KUKA KRL program: f1_Kuka_APT206T02S06.SRC

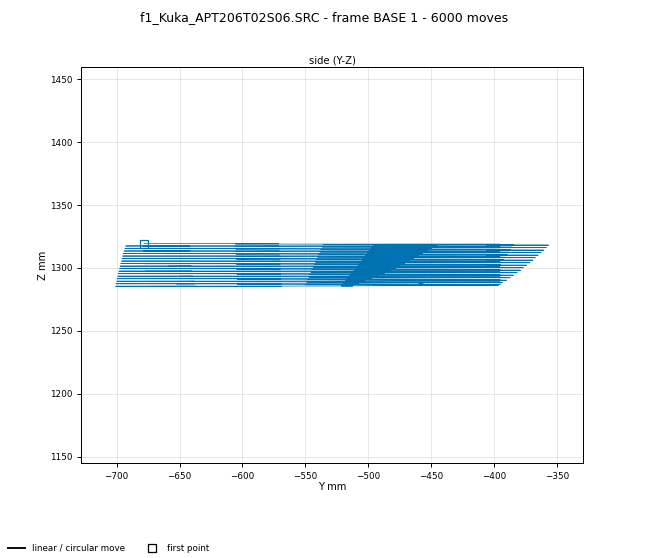
[picture p0: tool path of f1_Kuka_APT206T02S06.SRC in frame BASE 1, 6000 of 6001 moves have a stored position in this frame; points joined in program order, loops and branches not executed]
&ACCESS RVP
&REL 2
&PARAM TEMPLATE = C:\KRC\Roboter\Template\vorgabe
&PARAM EDITMASK = *
DEF f1_Kuka_APT206T02S06()


;FOLD INI;%{PE}%V3.2.0,%MKUKATPBASIS,%CINIT,%VCOMMON,%P
  ;FOLD BAS INI;%{E}%V3.2.0,%MKUKATPBASIS,%CINIT,%VINIT,%P
    GLOBAL INTERRUPT DECL 3 WHEN $STOPMESS==TRUE DO IR_STOPM ( )
    INTERRUPT ON 3
    BAS (#INITMOV,0 )
  ;ENDFOLD (BAS INI)
  ;FOLD USER INI;%{E}%V3.2.0,%MKUKATPUSER,%CINIT,%VINIT,%P
    ;Make your modifications here
  ;ENDFOLD (USER INI)
;ENDFOLD (INI)


;*** Make Null PTP Move
  PTP $pos_act

;*** Auto Load The Correct TOOL Data
  $tool=tool_data[2]

;*** Auto Load The Correct BASE Data
  $base=base_data[1]

  $ADVANCE = 5

;*** Restate Last Velocity
MMPM(30000.0)
SetRPM(8000)
LIN {X -0.383,Y -678.241,Z 1319.360,A 0.000,B 0.000,C 90.000,E1 100.782} C_DIS
LIN {X 0.191,Y -677.668,Z 1319.357,A 0.000,B 0.000,C 90.000,E1 100.254} C_DIS
LIN {X -0.027,Y -676.905,Z 1319.354,A 0.000,B 0.000,C 90.000,E1 99.792} C_DIS
LIN {X -0.134,Y -675.753,Z 1319.352,A 0.000,B 0.000,C 90.000,E1 99.321} C_DIS
LIN {X 0.307,Y -674.318,Z 1319.349,A 0.000,B 0.000,C 90.000,E1 98.803} C_DIS
LIN {X 0.076,Y -672.539,Z 1319.346,A 0.000,B 0.000,C 90.000,E1 98.341} C_DIS
LIN {X -0.071,Y -670.513,Z 1319.344,A 0.000,B 0.000,C 90.000,E1 97.871} C_DIS
LIN {X 0.337,Y -668.279,Z 1319.341,A 0.000,B 0.000,C 90.000,E1 97.352} C_DIS
LIN {X 0.069,Y -665.838,Z 1319.338,A 0.000,B 0.000,C 90.000,E1 96.891} C_DIS
LIN {X -0.309,Y -662.485,Z 1319.335,A 0.000,B 0.000,C 90.000,E1 96.315} C_DIS
LIN {X 0.043,Y -659.568,Z 1319.332,A 0.000,B 0.000,C 90.000,E1 95.796} C_DIS
LIN {X -0.281,Y -656.447,Z 1319.330,A 0.000,B 0.000,C 90.000,E1 95.334} C_DIS
LIN {X 0.072,Y -653.986,Z 1319.328,A 0.000,B 0.000,C 90.000,E1 94.935} C_DIS
LIN {X 0.254,Y -649.358,Z 1319.324,A 0.000,B 0.000,C 90.000,E1 94.302} C_DIS
LIN {X -0.138,Y -645.441,Z 1319.321,A 0.000,B 0.000,C 90.000,E1 93.841} C_DIS
LIN {X -0.068,Y -640.049,Z 1319.318,A 0.000,B 0.000,C 90.000,E1 93.212} C_DIS
LIN {X 0.118,Y -635.523,Z 1319.315,A 0.000,B 0.000,C 90.000,E1 92.694} C_DIS
LIN {X 0.245,Y -630.728,Z 1319.312,A 0.000,B 0.000,C 90.000,E1 92.178} C_DIS
LIN {X -0.245,Y -624.406,Z 1319.309,A 0.000,B 0.000,C 90.000,E1 91.604} C_DIS
LIN {X 0.064,Y -617.770,Z 1319.306,A 0.000,B 0.000,C 90.000,E1 90.974} C_DIS
LIN {X 0.019,Y -614.904,Z 1319.304,A 0.000,B 0.000,C 90.000,E1 90.745} C_DIS
LIN {X -0.082,Y -609.367,Z 1319.302,A 0.000,B 0.000,C 90.000,E1 90.344} C_DIS
LIN {X -0.088,Y -602.730,Z 1319.300,A 0.000,B 0.000,C 90.000,E1 89.943} C_DIS
LIN {X -0.187,Y -595.944,Z 1319.298,A 0.000,B 0.000,C 90.000,E1 89.599} C_DIS
LIN {X 0.165,Y -588.900,Z 1319.296,A 0.000,B 0.000,C 90.000,E1 89.255} C_DIS
LIN {X -0.024,Y -576.693,Z 1319.293,A 0.000,B 0.000,C 90.000,E1 88.797} C_DIS
LIN {X 0.193,Y -573.915,Z 1319.292,A 0.000,B 0.000,C 90.000,E1 88.625} C_DIS
LIN {X -0.066,Y -572.871,Z 1319.292,A 0.000,B 0.000,C 90.000,E1 88.568} C_DIS
LIN {X -0.103,Y -571.871,Z 1319.291,A 0.000,B 0.000,C 90.000,E1 88.453} C_DIS
LIN {X -0.146,Y -571.844,Z 1319.291,A 0.000,B 0.000,C 90.000,E1 88.453} C_DIS
LIN {X 0.218,Y -571.236,Z 1319.289,A 0.000,B 0.000,C 90.000,E1 88.051} C_DIS
LIN {X 0.134,Y -571.299,Z 1319.287,A 0.000,B 0.000,C 90.000,E1 87.650} C_DIS
LIN {X -0.010,Y -573.083,Z 1319.276,A 0.000,B 0.000,C 90.000,E1 85.755} C_DIS
LIN {X 0.263,Y -575.744,Z 1319.263,A 0.000,B 0.000,C 90.000,E1 83.280} C_DIS
LIN {X 0.201,Y -577.711,Z 1319.254,A 0.000,B 0.000,C 90.000,E1 81.659} C_DIS
LIN {X -0.044,Y -579.300,Z 1319.246,A 0.000,B 0.000,C 90.000,E1 80.330} C_DIS
LIN {X -0.175,Y -580.807,Z 1319.239,A 0.000,B 0.000,C 90.000,E1 78.993} C_DIS
LIN {X 0.169,Y -581.938,Z 1319.233,A 0.000,B 0.000,C 90.000,E1 77.881} C_DIS
LIN {X 0.193,Y -583.136,Z 1319.225,A 0.000,B 0.000,C 90.000,E1 76.533} C_DIS
LIN {X 0.043,Y -584.329,Z 1319.216,A 0.000,B 0.000,C 90.000,E1 74.936} C_DIS
LIN {X 0.076,Y -585.456,Z 1319.207,A 0.000,B 0.000,C 90.000,E1 73.323} C_DIS
LIN {X 0.230,Y -586.154,Z 1319.202,A 0.000,B 0.000,C 90.000,E1 72.236} C_DIS
LIN {X -0.261,Y -587.227,Z 1319.193,A 0.000,B 0.000,C 90.000,E1 70.678} C_DIS
LIN {X 0.165,Y -588.716,Z 1319.179,A 0.000,B 0.000,C 90.000,E1 68.230} C_DIS
LIN {X -0.209,Y -589.764,Z 1319.170,A 0.000,B 0.000,C 90.000,E1 66.666} C_DIS
LIN {X -0.020,Y -590.895,Z 1319.161,A 0.000,B 0.000,C 90.000,E1 65.049} C_DIS
LIN {X -0.038,Y -592.401,Z 1319.150,A 0.000,B 0.000,C 90.000,E1 62.922} C_DIS
LIN {X -0.001,Y -593.510,Z 1319.142,A 0.000,B 0.000,C 90.000,E1 61.591} C_DIS
LIN {X 0.096,Y -594.716,Z 1319.135,A 0.000,B 0.000,C 90.000,E1 60.255} C_DIS
LIN {X -0.078,Y -596.020,Z 1319.127,A 0.000,B 0.000,C 90.000,E1 58.948} C_DIS
LIN {X -0.312,Y -597.969,Z 1319.117,A 0.000,B 0.000,C 90.000,E1 57.120} C_DIS
LIN {X -0.311,Y -599.376,Z 1319.110,A 0.000,B 0.000,C 90.000,E1 55.801} C_DIS
LIN {X -0.284,Y -600.719,Z 1319.103,A 0.000,B 0.000,C 90.000,E1 54.482} C_DIS
LIN {X 0.114,Y -601.929,Z 1319.095,A 0.000,B 0.000,C 90.000,E1 53.130} C_DIS
LIN {X 0.055,Y -603.065,Z 1319.088,A 0.000,B 0.000,C 90.000,E1 51.823} C_DIS
LIN {X -0.244,Y -603.807,Z 1319.082,A 0.000,B 0.000,C 90.000,E1 50.803} C_DIS
LIN {X 0.106,Y -604.726,Z 1319.075,A 0.000,B 0.000,C 90.000,E1 49.461} C_DIS
LIN {X -0.043,Y -605.108,Z 1319.071,A 0.000,B 0.000,C 90.000,E1 48.690} C_DIS
LIN {X 0.066,Y -605.351,Z 1319.065,A 0.000,B 0.000,C 90.000,E1 47.634} C_DIS
LIN {X -0.002,Y -605.572,Z 1319.055,A 0.000,B 0.000,C 90.000,E1 45.810} C_DIS
LIN {X 0.276,Y -605.578,Z 1319.050,A 0.000,B 0.000,C 90.000,E1 45.000} C_DIS
LIN {X -0.029,Y -605.233,Z 1319.042,A 0.000,B 0.000,C 90.000,E1 43.461} C_DIS
LIN {X -0.319,Y -604.735,Z 1319.033,A 0.000,B 0.000,C 90.000,E1 41.919} C_DIS
LIN {X -0.415,Y -604.251,Z 1319.026,A 0.000,B 0.000,C 90.000,E1 40.620} C_DIS
LIN {X -0.018,Y -603.365,Z 1319.015,A 0.000,B 0.000,C 90.000,E1 38.749} C_DIS
LIN {X -0.317,Y -602.720,Z 1319.010,A 0.000,B 0.000,C 90.000,E1 37.729} C_DIS
LIN {X -0.036,Y -602.043,Z 1319.005,A 0.000,B 0.000,C 90.000,E1 36.916} C_DIS
LIN {X -0.126,Y -601.079,Z 1319.001,A 0.000,B 0.000,C 90.000,E1 36.137} C_DIS
LIN {X -0.086,Y -599.082,Z 1318.993,A 0.000,B 0.000,C 90.000,E1 34.818} C_DIS
LIN {X -0.077,Y -596.688,Z 1318.986,A 0.000,B 0.000,C 90.000,E1 33.499} C_DIS
LIN {X 0.269,Y -594.911,Z 1318.982,A 0.000,B 0.000,C 90.000,E1 32.673} C_DIS
LIN {X -0.331,Y -592.256,Z 1318.976,A 0.000,B 0.000,C 90.000,E1 31.671} C_DIS
LIN {X -0.233,Y -590.717,Z 1318.973,A 0.000,B 0.000,C 90.000,E1 31.131} C_DIS
LIN {X -0.261,Y -588.078,Z 1318.968,A 0.000,B 0.000,C 90.000,E1 30.335} C_DIS
LIN {X -0.314,Y -585.030,Z 1318.964,A 0.000,B 0.000,C 90.000,E1 29.539} C_DIS
LIN {X 0.236,Y -582.780,Z 1318.961,A 0.000,B 0.000,C 90.000,E1 28.949} C_DIS
LIN {X 0.121,Y -579.160,Z 1318.957,A 0.000,B 0.000,C 90.000,E1 28.153} C_DIS
LIN {X 0.202,Y -574.998,Z 1318.952,A 0.000,B 0.000,C 90.000,E1 27.334} C_DIS
LIN {X 0.073,Y -571.204,Z 1318.948,A 0.000,B 0.000,C 90.000,E1 26.668} C_DIS
LIN {X 0.163,Y -567.135,Z 1318.944,A 0.000,B 0.000,C 90.000,E1 25.976} C_DIS
LIN {X 0.219,Y -562.748,Z 1318.941,A 0.000,B 0.000,C 90.000,E1 25.283} C_DIS
LIN {X -0.269,Y -557.850,Z 1318.937,A 0.000,B 0.000,C 90.000,E1 24.643} C_DIS
LIN {X 0.063,Y -553.956,Z 1318.934,A 0.000,B 0.000,C 90.000,E1 24.079} C_DIS
LIN {X 0.002,Y -548.431,Z 1318.930,A 0.000,B 0.000,C 90.000,E1 23.387} C_DIS
LIN {X 0.018,Y -543.698,Z 1318.927,A 0.000,B 0.000,C 90.000,E1 22.823} C_DIS
LIN {X 0.077,Y -536.444,Z 1318.922,A 0.000,B 0.000,C 90.000,E1 21.972} C_DIS
LIN {X 0.048,Y -531.264,Z 1318.919,A 0.000,B 0.000,C 90.000,E1 21.408} C_DIS
LIN {X 0.199,Y -522.283,Z 1318.914,A 0.000,B 0.000,C 90.000,E1 20.429} C_DIS
LIN {X 0.149,Y -511.815,Z 1318.908,A 0.000,B 0.000,C 90.000,E1 19.341} C_DIS
LIN {X 0.057,Y -502.681,Z 1318.902,A 0.000,B 0.000,C 90.000,E1 18.417} C_DIS
LIN {X -0.001,Y -491.518,Z 1318.896,A 0.000,B 0.000,C 90.000,E1 17.330} C_DIS
LIN {X -0.041,Y -483.324,Z 1318.892,A 0.000,B 0.000,C 90.000,E1 16.551} C_DIS
LIN {X 0.178,Y -474.592,Z 1318.887,A 0.000,B 0.000,C 90.000,E1 15.717} C_DIS
LIN {X 0.167,Y -464.311,Z 1318.882,A 0.000,B 0.000,C 90.000,E1 14.773} C_DIS
LIN {X 0.215,Y -446.791,Z 1318.873,A 0.000,B 0.000,C 90.000,E1 13.119} C_DIS
LIN {X 0.151,Y -424.007,Z 1318.860,A 0.000,B 0.000,C 90.000,E1 10.782} C_DIS
LIN {X 0.086,Y -406.860,Z 1318.850,A 0.000,B 0.000,C 90.000,E1 8.916} C_DIS
LIN {X -0.204,Y -398.311,Z 1318.844,A 0.000,B 0.000,C 90.000,E1 7.992} C_DIS
LIN {X -0.085,Y -395.321,Z 1318.842,A 0.000,B 0.000,C 90.000,E1 7.530} C_DIS
LIN {X -0.124,Y -395.315,Z 1318.842,A 0.000,B 0.000,C 90.000,E1 7.530} C_DIS
LIN {X 0.155,Y -395.949,Z 1318.841,A 0.000,B 0.000,C 90.000,E1 7.352} C_DIS
LIN {X 0.118,Y -395.998,Z 1318.841,A 0.000,B 0.000,C 90.000,E1 7.352} C_DIS
LIN {X -0.054,Y -399.469,Z 1318.839,A 0.000,B 0.000,C 90.000,E1 7.068} C_DIS
LIN {X 0.042,Y -405.000,Z 1318.837,A 0.000,B 0.000,C 90.000,E1 6.663} C_DIS
LIN {X 0.063,Y -409.735,Z 1318.835,A 0.000,B 0.000,C 90.000,E1 6.372} C_DIS
LIN {X 0.004,Y -417.825,Z 1318.833,A 0.000,B 0.000,C 90.000,E1 5.853} C_DIS
LIN {X 0.038,Y -424.124,Z 1318.830,A 0.000,B 0.000,C 90.000,E1 5.391} C_DIS
LIN {X -0.173,Y -430.359,Z 1318.827,A 0.000,B 0.000,C 90.000,E1 4.935} C_DIS
LIN {X -0.043,Y -439.367,Z 1318.823,A 0.000,B 0.000,C 90.000,E1 4.131} C_DIS
LIN {X -0.035,Y -443.739,Z 1318.821,A 0.000,B 0.000,C 90.000,E1 3.726} C_DIS
LIN {X 0.021,Y -449.647,Z 1318.818,A 0.000,B 0.000,C 90.000,E1 3.154} C_DIS
LIN {X 0.047,Y -455.368,Z 1318.814,A 0.000,B 0.000,C 90.000,E1 2.579} C_DIS
LIN {X -0.123,Y -460.898,Z 1318.811,A 0.000,B 0.000,C 90.000,E1 2.007} C_DIS
LIN {X 0.217,Y -467.528,Z 1318.807,A 0.000,B 0.000,C 90.000,E1 1.203} C_DIS
LIN {X -0.216,Y -472.449,Z 1318.803,A 0.000,B 0.000,C 90.000,E1 0.630} C_DIS
LIN {X 0.000,Y -476.981,Z 1318.800,A 0.000,B 0.000,C 90.000,E1 360.000} C_DIS
LIN {X 0.121,Y -481.653,Z 1318.796,A 0.000,B 0.000,C 90.000,E1 359.312} C_DIS
LIN {X -0.103,Y -486.586,Z 1318.792,A 0.000,B 0.000,C 90.000,E1 358.568} C_DIS
LIN {X 0.222,Y -491.172,Z 1318.788,A 0.000,B 0.000,C 90.000,E1 357.764} C_DIS
LIN {X 0.081,Y -495.438,Z 1318.784,A 0.000,B 0.000,C 90.000,E1 357.020} C_DIS
LIN {X -0.179,Y -498.630,Z 1318.780,A 0.000,B 0.000,C 90.000,E1 356.445} C_DIS
LIN {X -0.041,Y -503.078,Z 1318.775,A 0.000,B 0.000,C 90.000,E1 355.527} C_DIS
LIN {X -0.048,Y -506.551,Z 1318.771,A 0.000,B 0.000,C 90.000,E1 354.780} C_DIS
LIN {X -0.078,Y -511.007,Z 1318.765,A 0.000,B 0.000,C 90.000,E1 353.742} C_DIS
LIN {X -0.226,Y -513.361,Z 1318.762,A 0.000,B 0.000,C 90.000,E1 353.166} C_DIS
LIN {X 0.122,Y -516.546,Z 1318.757,A 0.000,B 0.000,C 90.000,E1 352.243} C_DIS
LIN {X -0.006,Y -519.467,Z 1318.752,A 0.000,B 0.000,C 90.000,E1 351.376} C_DIS
LIN {X -0.022,Y -521.276,Z 1318.749,A 0.000,B 0.000,C 90.000,E1 350.792} C_DIS
LIN {X -0.103,Y -523.788,Z 1318.744,A 0.000,B 0.000,C 90.000,E1 349.926} C_DIS
LIN {X -0.068,Y -526.011,Z 1318.739,A 0.000,B 0.000,C 90.000,E1 349.050} C_DIS
LIN {X 0.018,Y -528.682,Z 1318.733,A 0.000,B 0.000,C 90.000,E1 347.881} C_DIS
LIN {X 0.225,Y -530.374,Z 1318.728,A 0.000,B 0.000,C 90.000,E1 346.992} C_DIS
LIN {X -0.184,Y -531.781,Z 1318.723,A 0.000,B 0.000,C 90.000,E1 346.172} C_DIS
LIN {X 0.104,Y -533.446,Z 1318.717,A 0.000,B 0.000,C 90.000,E1 344.991} C_DIS
LIN {X -0.145,Y -534.384,Z 1318.712,A 0.000,B 0.000,C 90.000,E1 344.157} C_DIS
LIN {X 0.130,Y -535.065,Z 1318.707,A 0.000,B 0.000,C 90.000,E1 343.268} C_DIS
LIN {X 0.055,Y -535.458,Z 1318.702,A 0.000,B 0.000,C 90.000,E1 342.417} C_DIS
LIN {X -0.177,Y -535.659,Z 1318.698,A 0.000,B 0.000,C 90.000,E1 341.583} C_DIS
LIN {X -0.239,Y -535.454,Z 1318.693,A 0.000,B 0.000,C 90.000,E1 340.732} C_DIS
LIN {X -0.094,Y -534.784,Z 1318.687,A 0.000,B 0.000,C 90.000,E1 339.571} C_DIS
LIN {X 0.128,Y -534.219,Z 1318.683,A 0.000,B 0.000,C 90.000,E1 338.975} C_DIS
LIN {X 0.240,Y -533.293,Z 1318.679,A 0.000,B 0.000,C 90.000,E1 338.103} C_DIS
LIN {X -0.053,Y -532.872,Z 1318.677,A 0.000,B 0.000,C 90.000,E1 337.847} C_DIS
LIN {X 0.051,Y -531.324,Z 1318.672,A 0.000,B 0.000,C 90.000,E1 336.975} C_DIS
LIN {X -0.157,Y -528.693,Z 1318.666,A 0.000,B 0.000,C 90.000,E1 335.845} C_DIS
LIN {X 0.205,Y -527.147,Z 1318.663,A 0.000,B 0.000,C 90.000,E1 335.229} C_DIS
LIN {X -0.235,Y -524.541,Z 1318.658,A 0.000,B 0.000,C 90.000,E1 334.409} C_DIS
LIN {X 0.059,Y -519.924,Z 1318.650,A 0.000,B 0.000,C 90.000,E1 332.922} C_DIS
LIN {X 0.023,Y -515.240,Z 1318.641,A 0.000,B 0.000,C 90.000,E1 331.463} C_DIS
LIN {X 0.037,Y -511.177,Z 1318.635,A 0.000,B 0.000,C 90.000,E1 330.284} C_DIS
LIN {X -0.085,Y -508.003,Z 1318.630,A 0.000,B 0.000,C 90.000,E1 329.410} C_DIS
LIN {X 0.080,Y -503.370,Z 1318.623,A 0.000,B 0.000,C 90.000,E1 328.201} C_DIS
LIN {X -0.250,Y -498.639,Z 1318.617,A 0.000,B 0.000,C 90.000,E1 327.041} C_DIS
LIN {X 0.183,Y -495.521,Z 1318.612,A 0.000,B 0.000,C 90.000,E1 326.087} C_DIS
LIN {X 0.167,Y -492.720,Z 1318.607,A 0.000,B 0.000,C 90.000,E1 325.182} C_DIS
LIN {X -0.127,Y -491.111,Z 1318.603,A 0.000,B 0.000,C 90.000,E1 324.609} C_DIS
LIN {X -0.033,Y -489.329,Z 1318.600,A 0.000,B 0.000,C 90.000,E1 323.989} C_DIS
LIN {X -0.125,Y -487.674,Z 1318.597,A 0.000,B 0.000,C 90.000,E1 323.543} C_DIS
LIN {X 0.104,Y -486.223,Z 1318.596,A 0.000,B 0.000,C 90.000,E1 323.210} C_DIS
LIN {X 0.167,Y -485.215,Z 1318.595,A 0.000,B 0.000,C 90.000,E1 323.050} C_DIS
LIN {X -0.037,Y -480.453,Z 1318.592,A 0.000,B 0.000,C 90.000,E1 322.637} C_DIS
LIN {X -0.028,Y -458.983,Z 1318.581,A 0.000,B 0.000,C 90.000,E1 320.598} C_DIS
LIN {X -0.036,Y -438.160,Z 1318.569,A 0.000,B 0.000,C 90.000,E1 318.366} C_DIS
LIN {X 0.243,Y -419.408,Z 1318.556,A 0.000,B 0.000,C 90.000,E1 316.053} C_DIS
LIN {X -0.126,Y -401.927,Z 1318.543,A 0.000,B 0.000,C 90.000,E1 313.704} C_DIS
LIN {X -0.083,Y -386.080,Z 1318.529,A 0.000,B 0.000,C 90.000,E1 311.229} C_DIS
LIN {X 0.007,Y -384.707,Z 1318.528,A 0.000,B 0.000,C 90.000,E1 310.987} C_DIS
LIN {X -0.031,Y -384.677,Z 1318.528,A 0.000,B 0.000,C 90.000,E1 310.987} C_DIS
LIN {X -0.095,Y -385.211,Z 1318.524,A 0.000,B 0.000,C 90.000,E1 310.334} C_DIS
LIN {X -0.129,Y -391.258,Z 1318.492,A 0.000,B 0.000,C 90.000,E1 304.612} C_DIS
LIN {X 0.025,Y -396.971,Z 1318.459,A 0.000,B 0.000,C 90.000,E1 298.565} C_DIS
LIN {X -0.024,Y -401.336,Z 1318.427,A 0.000,B 0.000,C 90.000,E1 292.950} C_DIS
LIN {X 0.056,Y -401.655,Z 1318.426,A 0.000,B 0.000,C 90.000,E1 292.589} C_DIS
LIN {X -0.178,Y -404.743,Z 1318.395,A 0.000,B 0.000,C 90.000,E1 287.040} C_DIS
LIN {X -0.176,Y -406.153,Z 1318.364,A 0.000,B 0.000,C 90.000,E1 281.478} C_DIS
LIN {X -0.077,Y -405.680,Z 1318.333,A 0.000,B 0.000,C 90.000,E1 275.910} C_DIS
LIN {X -0.006,Y -403.567,Z 1318.306,A 0.000,B 0.000,C 90.000,E1 271.031} C_DIS
LIN {X -0.071,Y -403.188,Z 1318.302,A 0.000,B 0.000,C 90.000,E1 270.344} C_DIS
LIN {X 0.163,Y -399.069,Z 1318.273,A 0.000,B 0.000,C 90.000,E1 265.065} C_DIS
LIN {X 0.104,Y -398.785,Z 1318.271,A 0.000,B 0.000,C 90.000,E1 264.723} C_DIS
LIN {X -0.006,Y -393.297,Z 1318.243,A 0.000,B 0.000,C 90.000,E1 259.803} C_DIS
LIN {X -0.085,Y -392.681,Z 1318.240,A 0.000,B 0.000,C 90.000,E1 259.106} C_DIS
LIN {X 0.085,Y -386.254,Z 1318.214,A 0.000,B 0.000,C 90.000,E1 254.448} C_DIS
LIN {X 0.050,Y -385.156,Z 1318.208,A 0.000,B 0.000,C 90.000,E1 253.378} C_DIS
LIN {X -0.194,Y -377.824,Z 1318.182,A 0.000,B 0.000,C 90.000,E1 248.720} C_DIS
LIN {X 0.030,Y -376.094,Z 1318.174,A 0.000,B 0.000,C 90.000,E1 247.230} C_DIS
LIN {X 0.087,Y -368.762,Z 1318.149,A 0.000,B 0.000,C 90.000,E1 242.820} C_DIS
LIN {X 0.071,Y -366.406,Z 1318.139,A 0.000,B 0.000,C 90.000,E1 240.973} C_DIS
LIN {X -0.080,Y -365.114,Z 1318.135,A 0.000,B 0.000,C 90.000,E1 240.255} C_DIS
LIN {X -0.015,Y -358.513,Z 1318.112,A 0.000,B 0.000,C 90.000,E1 236.135} C_DIS
LIN {X 0.183,Y -356.725,Z 1318.104,A 0.000,B 0.000,C 90.000,E1 234.689} C_DIS
LIN {X 0.164,Y -356.733,Z 1318.104,A 0.000,B 0.000,C 90.000,E1 234.689} C_DIS
LIN {X 0.149,Y -369.901,Z 1318.089,A 0.000,B 0.000,C 90.000,E1 231.984} C_DIS
LIN {X -0.088,Y -384.084,Z 1318.075,A 0.000,B 0.000,C 90.000,E1 229.461} C_DIS
LIN {X 0.051,Y -399.786,Z 1318.061,A 0.000,B 0.000,C 90.000,E1 226.944} C_DIS
LIN {X 0.060,Y -417.123,Z 1318.047,A 0.000,B 0.000,C 90.000,E1 224.514} C_DIS
LIN {X -0.143,Y -436.025,Z 1318.034,A 0.000,B 0.000,C 90.000,E1 222.204} C_DIS
LIN {X 0.039,Y -442.970,Z 1318.030,A 0.000,B 0.000,C 90.000,E1 221.391} C_DIS
LIN {X 0.086,Y -444.000,Z 1318.029,A 0.000,B 0.000,C 90.000,E1 221.229} C_DIS
LIN {X 0.072,Y -444.740,Z 1318.028,A 0.000,B 0.000,C 90.000,E1 221.067} C_DIS
LIN {X 0.057,Y -445.323,Z 1318.027,A 0.000,B 0.000,C 90.000,E1 220.906} C_DIS
LIN {X -0.257,Y -446.232,Z 1318.026,A 0.000,B 0.000,C 90.000,E1 220.620} C_DIS
LIN {X 0.041,Y -447.543,Z 1318.022,A 0.000,B 0.000,C 90.000,E1 219.930} C_DIS
LIN {X 0.047,Y -448.891,Z 1318.016,A 0.000,B 0.000,C 90.000,E1 218.955} C_DIS
LIN {X -0.213,Y -449.860,Z 1318.011,A 0.000,B 0.000,C 90.000,E1 218.016} C_DIS
LIN {X 0.004,Y -451.726,Z 1317.999,A 0.000,B 0.000,C 90.000,E1 215.724} C_DIS
LIN {X 0.036,Y -454.835,Z 1317.981,A 0.000,B 0.000,C 90.000,E1 212.498} C_DIS
LIN {X 0.106,Y -457.731,Z 1317.966,A 0.000,B 0.000,C 90.000,E1 209.922} C_DIS
LIN {X -0.054,Y -460.143,Z 1317.956,A 0.000,B 0.000,C 90.000,E1 208.025} C_DIS
LIN {X -0.041,Y -463.318,Z 1317.943,A 0.000,B 0.000,C 90.000,E1 205.796} C_DIS
LIN {X -0.003,Y -465.641,Z 1317.935,A 0.000,B 0.000,C 90.000,E1 204.207} C_DIS
LIN {X -0.062,Y -467.436,Z 1317.927,A 0.000,B 0.000,C 90.000,E1 202.950} C_DIS
LIN {X 0.159,Y -469.187,Z 1317.921,A 0.000,B 0.000,C 90.000,E1 201.663} C_DIS
LIN {X -0.156,Y -472.148,Z 1317.908,A 0.000,B 0.000,C 90.000,E1 199.504} C_DIS
LIN {X 0.175,Y -475.170,Z 1317.896,A 0.000,B 0.000,C 90.000,E1 197.275} C_DIS
LIN {X 0.023,Y -477.737,Z 1317.886,A 0.000,B 0.000,C 90.000,E1 195.426} C_DIS
LIN {X -0.199,Y -480.198,Z 1317.875,A 0.000,B 0.000,C 90.000,E1 193.592} C_DIS
LIN {X -0.143,Y -483.051,Z 1317.863,A 0.000,B 0.000,C 90.000,E1 191.422} C_DIS
LIN {X 0.148,Y -485.080,Z 1317.855,A 0.000,B 0.000,C 90.000,E1 189.849} C_DIS
LIN {X 0.155,Y -487.890,Z 1317.843,A 0.000,B 0.000,C 90.000,E1 187.701} C_DIS
LIN {X 0.086,Y -489.358,Z 1317.836,A 0.000,B 0.000,C 90.000,E1 186.486} C_DIS
LIN {X 0.181,Y -491.417,Z 1317.826,A 0.000,B 0.000,C 90.000,E1 184.645} C_DIS
LIN {X 0.073,Y -492.529,Z 1317.819,A 0.000,B 0.000,C 90.000,E1 183.440} C_DIS
LIN {X -0.162,Y -493.843,Z 1317.811,A 0.000,B 0.000,C 90.000,E1 181.949} C_DIS
LIN {X -0.090,Y -494.487,Z 1317.806,A 0.000,B 0.000,C 90.000,E1 181.031} C_DIS
LIN {X 0.190,Y -495.305,Z 1317.797,A 0.000,B 0.000,C 90.000,E1 179.484} C_DIS
LIN {X -0.231,Y -495.590,Z 1317.792,A 0.000,B 0.000,C 90.000,E1 178.625} C_DIS
LIN {X -0.139,Y -495.793,Z 1317.787,A 0.000,B 0.000,C 90.000,E1 177.707} C_DIS
LIN {X 0.170,Y -495.635,Z 1317.779,A 0.000,B 0.000,C 90.000,E1 176.159} C_DIS
LIN {X 0.156,Y -495.070,Z 1317.772,A 0.000,B 0.000,C 90.000,E1 174.951} C_DIS
LIN {X -0.252,Y -494.459,Z 1317.767,A 0.000,B 0.000,C 90.000,E1 174.090} C_DIS
LIN {X -0.125,Y -493.637,Z 1317.762,A 0.000,B 0.000,C 90.000,E1 173.166} C_DIS
LIN {X -0.006,Y -492.635,Z 1317.757,A 0.000,B 0.000,C 90.000,E1 172.243} C_DIS
LIN {X -0.212,Y -491.801,Z 1317.754,A 0.000,B 0.000,C 90.000,E1 171.659} C_DIS
LIN {X -0.222,Y -489.624,Z 1317.747,A 0.000,B 0.000,C 90.000,E1 170.443} C_DIS
LIN {X -0.072,Y -487.714,Z 1317.742,A 0.000,B 0.000,C 90.000,E1 169.511} C_DIS
LIN {X 0.055,Y -485.335,Z 1317.737,A 0.000,B 0.000,C 90.000,E1 168.578} C_DIS
LIN {X -0.191,Y -483.563,Z 1317.733,A 0.000,B 0.000,C 90.000,E1 167.993} C_DIS
LIN {X -0.118,Y -480.351,Z 1317.728,A 0.000,B 0.000,C 90.000,E1 167.061} C_DIS
LIN {X -0.148,Y -479.211,Z 1317.726,A 0.000,B 0.000,C 90.000,E1 166.756} C_DIS
LIN {X 0.070,Y -473.871,Z 1317.720,A 0.000,B 0.000,C 90.000,E1 165.644} C_DIS
LIN {X -0.132,Y -467.316,Z 1317.714,A 0.000,B 0.000,C 90.000,E1 164.574} C_DIS
LIN {X -0.210,Y -454.598,Z 1317.702,A 0.000,B 0.000,C 90.000,E1 162.362} C_DIS
LIN {X 0.166,Y -450.662,Z 1317.698,A 0.000,B 0.000,C 90.000,E1 161.511} C_DIS
LIN {X -0.064,Y -447.559,Z 1317.693,A 0.000,B 0.000,C 90.000,E1 160.732} C_DIS
LIN {X -0.170,Y -446.128,Z 1317.688,A 0.000,B 0.000,C 90.000,E1 159.934} C_DIS
LIN {X -0.102,Y -446.821,Z 1317.686,A 0.000,B 0.000,C 90.000,E1 159.444} C_DIS
LIN {X 0.187,Y -448.646,Z 1317.684,A 0.000,B 0.000,C 90.000,E1 159.082} C_DIS
LIN {X -0.031,Y -449.305,Z 1317.683,A 0.000,B 0.000,C 90.000,E1 159.028} C_DIS
LIN {X 0.043,Y -460.836,Z 1317.678,A 0.000,B 0.000,C 90.000,E1 158.028} C_DIS
LIN {X 0.256,Y -476.353,Z 1317.671,A 0.000,B 0.000,C 90.000,E1 156.794} C_DIS
LIN {X -0.097,Y -485.313,Z 1317.667,A 0.000,B 0.000,C 90.000,E1 156.102} C_DIS
LIN {X -0.035,Y -489.810,Z 1317.665,A 0.000,B 0.000,C 90.000,E1 155.717} C_DIS
LIN {X 0.068,Y -496.855,Z 1317.661,A 0.000,B 0.000,C 90.000,E1 155.049} C_DIS
LIN {X -0.198,Y -502.380,Z 1317.658,A 0.000,B 0.000,C 90.000,E1 154.537} C_DIS
LIN {X -0.035,Y -506.447,Z 1317.656,A 0.000,B 0.000,C 90.000,E1 154.101} C_DIS
LIN {X 0.003,Y -513.977,Z 1317.651,A 0.000,B 0.000,C 90.000,E1 153.256} C_DIS
LIN {X -0.021,Y -517.631,Z 1317.649,A 0.000,B 0.000,C 90.000,E1 152.820} C_DIS
LIN {X -0.124,Y -520.007,Z 1317.647,A 0.000,B 0.000,C 90.000,E1 152.538} C_DIS
LIN {X -0.074,Y -524.176,Z 1317.644,A 0.000,B 0.000,C 90.000,E1 151.948} C_DIS
LIN {X -0.245,Y -527.927,Z 1317.641,A 0.000,B 0.000,C 90.000,E1 151.385} C_DIS
LIN {X -0.289,Y -531.708,Z 1317.637,A 0.000,B 0.000,C 90.000,E1 150.667} C_DIS
LIN {X -0.038,Y -534.635,Z 1317.633,A 0.000,B 0.000,C 90.000,E1 149.921} C_DIS
LIN {X 0.116,Y -536.668,Z 1317.630,A 0.000,B 0.000,C 90.000,E1 149.331} C_DIS
LIN {X 0.000,Y -539.012,Z 1317.625,A 0.000,B 0.000,C 90.000,E1 148.486} C_DIS
LIN {X 0.007,Y -540.329,Z 1317.622,A 0.000,B 0.000,C 90.000,E1 147.916} C_DIS
LIN {X 0.213,Y -541.915,Z 1317.617,A 0.000,B 0.000,C 90.000,E1 147.041} C_DIS
LIN {X -0.044,Y -542.832,Z 1317.614,A 0.000,B 0.000,C 90.000,E1 146.501} C_DIS
LIN {X -0.208,Y -544.612,Z 1317.606,A 0.000,B 0.000,C 90.000,E1 145.102} C_DIS
LIN {X -0.300,Y -546.399,Z 1317.597,A 0.000,B 0.000,C 90.000,E1 143.417} C_DIS
LIN {X -0.216,Y -546.997,Z 1317.594,A 0.000,B 0.000,C 90.000,E1 142.844} C_DIS
LIN {X -0.173,Y -547.502,Z 1317.592,A 0.000,B 0.000,C 90.000,E1 142.557} C_DIS
LIN {X 0.063,Y -548.045,Z 1317.590,A 0.000,B 0.000,C 90.000,E1 142.110} C_DIS
LIN {X 0.244,Y -548.863,Z 1317.588,A 0.000,B 0.000,C 90.000,E1 141.823} C_DIS
LIN {X 0.200,Y -548.916,Z 1317.588,A 0.000,B 0.000,C 90.000,E1 141.823} C_DIS
LIN {X -0.034,Y -551.756,Z 1317.587,A 0.000,B 0.000,C 90.000,E1 141.698} C_DIS
LIN {X -0.093,Y -553.743,Z 1317.587,A 0.000,B 0.000,C 90.000,E1 141.618} C_DIS
LIN {X 0.094,Y -563.331,Z 1317.585,A 0.000,B 0.000,C 90.000,E1 141.295} C_DIS
LIN {X 0.262,Y -566.452,Z 1317.584,A 0.000,B 0.000,C 90.000,E1 141.170} C_DIS
LIN {X -0.097,Y -569.293,Z 1317.584,A 0.000,B 0.000,C 90.000,E1 141.090} C_DIS
LIN {X -0.204,Y -575.437,Z 1317.582,A 0.000,B 0.000,C 90.000,E1 140.803} C_DIS
LIN {X -0.236,Y -578.438,Z 1317.581,A 0.000,B 0.000,C 90.000,E1 140.642} C_DIS
LIN {X 0.054,Y -581.401,Z 1317.580,A 0.000,B 0.000,C 90.000,E1 140.436} C_DIS
LIN {X -0.223,Y -584.251,Z 1317.579,A 0.000,B 0.000,C 90.000,E1 140.275} C_DIS
LIN {X 0.033,Y -589.720,Z 1317.577,A 0.000,B 0.000,C 90.000,E1 139.828} C_DIS
LIN {X 0.284,Y -593.820,Z 1317.575,A 0.000,B 0.000,C 90.000,E1 139.461} C_DIS
LIN {X -0.123,Y -598.995,Z 1317.572,A 0.000,B 0.000,C 90.000,E1 139.013} C_DIS
LIN {X 0.148,Y -603.528,Z 1317.570,A 0.000,B 0.000,C 90.000,E1 138.528} C_DIS
LIN {X 0.080,Y -606.877,Z 1317.568,A 0.000,B 0.000,C 90.000,E1 138.162} C_DIS
LIN {X -0.030,Y -611.942,Z 1317.564,A 0.000,B 0.000,C 90.000,E1 137.553} C_DIS
LIN {X 0.066,Y -615.967,Z 1317.561,A 0.000,B 0.000,C 90.000,E1 137.025} C_DIS
LIN {X -0.261,Y -619.773,Z 1317.558,A 0.000,B 0.000,C 90.000,E1 136.539} C_DIS
LIN {X 0.177,Y -624.946,Z 1317.554,A 0.000,B 0.000,C 90.000,E1 135.729} C_DIS
LIN {X -0.334,Y -631.425,Z 1317.549,A 0.000,B 0.000,C 90.000,E1 134.757} C_DIS
LIN {X 0.337,Y -634.527,Z 1317.546,A 0.000,B 0.000,C 90.000,E1 134.190} C_DIS
LIN {X 0.036,Y -639.057,Z 1317.542,A 0.000,B 0.000,C 90.000,E1 133.461} C_DIS
LIN {X 0.163,Y -644.766,Z 1317.536,A 0.000,B 0.000,C 90.000,E1 132.447} C_DIS
LIN {X -0.122,Y -651.098,Z 1317.530,A 0.000,B 0.000,C 90.000,E1 131.353} C_DIS
LIN {X -0.222,Y -655.223,Z 1317.526,A 0.000,B 0.000,C 90.000,E1 130.620} C_DIS
LIN {X 0.172,Y -659.837,Z 1317.521,A 0.000,B 0.000,C 90.000,E1 129.725} C_DIS
LIN {X -0.312,Y -664.178,Z 1317.516,A 0.000,B 0.000,C 90.000,E1 128.910} C_DIS
LIN {X 0.208,Y -669.848,Z 1317.509,A 0.000,B 0.000,C 90.000,E1 127.649} C_DIS
LIN {X -0.115,Y -672.849,Z 1317.505,A 0.000,B 0.000,C 90.000,E1 126.950} C_DIS
LIN {X -0.004,Y -675.542,Z 1317.501,A 0.000,B 0.000,C 90.000,E1 126.217} C_DIS
LIN {X -0.270,Y -678.049,Z 1317.497,A 0.000,B 0.000,C 90.000,E1 125.518} C_DIS
LIN {X 0.048,Y -680.361,Z 1317.493,A 0.000,B 0.000,C 90.000,E1 124.771} C_DIS
LIN {X -0.167,Y -682.448,Z 1317.489,A 0.000,B 0.000,C 90.000,E1 124.072} C_DIS
LIN {X -0.364,Y -684.322,Z 1317.485,A 0.000,B 0.000,C 90.000,E1 123.372} C_DIS
LIN {X 0.026,Y -685.970,Z 1317.481,A 0.000,B 0.000,C 90.000,E1 122.625} C_DIS
LIN {X -0.149,Y -687.441,Z 1317.477,A 0.000,B 0.000,C 90.000,E1 121.926} C_DIS
LIN {X -0.458,Y -689.174,Z 1317.472,A 0.000,B 0.000,C 90.000,E1 121.003} C_DIS
LIN {X -0.025,Y -690.257,Z 1317.468,A 0.000,B 0.000,C 90.000,E1 120.256} C_DIS
LIN {X -0.061,Y -691.772,Z 1317.462,A 0.000,B 0.000,C 90.000,E1 119.077} C_DIS
LIN {X 0.052,Y -692.297,Z 1317.458,A 0.000,B 0.000,C 90.000,E1 118.359} C_DIS
LIN {X 0.414,Y -692.731,Z 1317.452,A 0.000,B 0.000,C 90.000,E1 117.385} C_DIS
LIN {X -0.153,Y -692.855,Z 1317.447,A 0.000,B 0.000,C 90.000,E1 116.488} C_DIS
LIN {X 0.339,Y -692.758,Z 1317.444,A 0.000,B 0.000,C 90.000,E1 115.976} C_DIS
LIN {X 0.151,Y -692.312,Z 1317.441,A 0.000,B 0.000,C 90.000,E1 115.283} C_DIS
LIN {X -0.231,Y -692.113,Z 1317.439,A 0.000,B 0.000,C 90.000,E1 115.079} C_DIS
LIN {X -0.038,Y -691.442,Z 1317.437,A 0.000,B 0.000,C 90.000,E1 114.591} C_DIS
LIN {X 0.203,Y -690.925,Z 1317.435,A 0.000,B 0.000,C 90.000,E1 114.335} C_DIS
LIN {X -0.234,Y -689.543,Z 1317.433,A 0.000,B 0.000,C 90.000,E1 113.898} C_DIS
LIN {X 0.348,Y -686.399,Z 1317.429,A 0.000,B 0.000,C 90.000,E1 113.259} C_DIS
LIN {X 0.199,Y -685.478,Z 1317.429,A 0.000,B 0.000,C 90.000,E1 113.153} C_DIS
LIN {X -0.065,Y -680.370,Z 1317.426,A 0.000,B 0.000,C 90.000,E1 112.717} C_DIS
LIN {X 0.091,Y -678.702,Z 1317.426,A 0.000,B 0.000,C 90.000,E1 112.589} C_DIS
LIN {X 0.036,Y -674.213,Z 1317.425,A 0.000,B 0.000,C 90.000,E1 112.408} C_DIS
LIN {X 0.084,Y -671.779,Z 1317.424,A 0.000,B 0.000,C 90.000,E1 112.333} C_DIS
LIN {X 0.391,Y -668.977,Z 1317.424,A 0.000,B 0.000,C 90.000,E1 112.206} C_DIS
LIN {X -0.146,Y -665.460,Z 1317.423,A 0.000,B 0.000,C 90.000,E1 112.153} C_DIS
LIN {X -0.093,Y -657.230,Z 1317.422,A 0.000,B 0.000,C 90.000,E1 112.025} C_DIS
LIN {X -0.181,Y -649.417,Z 1317.422,A 0.000,B 0.000,C 90.000,E1 111.972} C_DIS
LIN {X -0.143,Y -643.804,Z 1317.422,A 0.000,B 0.000,C 90.000,E1 111.897} C_DIS
LIN {X -0.165,Y -642.180,Z 1317.421,A 0.000,B 0.000,C 90.000,E1 111.844} C_DIS
LIN {X -0.207,Y -642.170,Z 1317.421,A 0.000,B 0.000,C 90.000,E1 111.844} C_DIS
LIN {X 0.355,Y -643.212,Z 1317.420,A 0.000,B 0.000,C 90.000,E1 111.589} C_DIS
LIN {X 0.246,Y -647.261,Z 1317.417,A 0.000,B 0.000,C 90.000,E1 111.099} C_DIS
LIN {X 0.200,Y -652.016,Z 1317.414,A 0.000,B 0.000,C 90.000,E1 110.482} C_DIS
LIN {X -0.032,Y -656.193,Z 1317.411,A 0.000,B 0.000,C 90.000,E1 109.885} C_DIS
LIN {X -0.009,Y -659.838,Z 1317.407,A 0.000,B 0.000,C 90.000,E1 109.268} C_DIS
LIN {X -0.119,Y -663.485,Z 1317.403,A 0.000,B 0.000,C 90.000,E1 108.544} C_DIS
LIN {X -0.200,Y -666.611,Z 1317.399,A 0.000,B 0.000,C 90.000,E1 107.819} C_DIS
LIN {X -0.171,Y -668.503,Z 1317.396,A 0.000,B 0.000,C 90.000,E1 107.330} C_DIS
LIN {X 0.240,Y -670.988,Z 1317.392,A 0.000,B 0.000,C 90.000,E1 106.567} C_DIS
LIN {X 0.293,Y -672.513,Z 1317.390,A 0.000,B 0.000,C 90.000,E1 106.079} C_DIS
LIN {X 0.109,Y -674.366,Z 1317.385,A 0.000,B 0.000,C 90.000,E1 105.371} C_DIS
LIN {X -0.053,Y -675.912,Z 1317.381,A 0.000,B 0.000,C 90.000,E1 104.662} C_DIS
LIN {X -0.083,Y -677.612,Z 1317.376,A 0.000,B 0.000,C 90.000,E1 103.703} C_DIS
LIN {X -0.375,Y -678.345,Z 1317.372,A 0.000,B 0.000,C 90.000,E1 103.008} C_DIS
LIN {X 0.163,Y -678.722,Z 1317.368,A 0.000,B 0.000,C 90.000,E1 102.243} C_DIS
LIN {X 0.077,Y -678.790,Z 1317.365,A 0.000,B 0.000,C 90.000,E1 101.771} C_DIS
LIN {X -0.010,Y -678.660,Z 1317.363,A 0.000,B 0.000,C 90.000,E1 101.299} C_DIS
LIN {X -0.275,Y -678.057,Z 1317.359,A 0.000,B 0.000,C 90.000,E1 100.602} C_DIS
LIN {X 0.294,Y -677.404,Z 1317.356,A 0.000,B 0.000,C 90.000,E1 100.074} C_DIS
LIN {X 0.126,Y -677.036,Z 1317.355,A 0.000,B 0.000,C 90.000,E1 99.849} C_DIS
LIN {X 0.018,Y -675.949,Z 1317.352,A 0.000,B 0.000,C 90.000,E1 99.378} C_DIS
LIN {X -0.208,Y -674.562,Z 1317.349,A 0.000,B 0.000,C 90.000,E1 98.916} C_DIS
LIN {X -0.272,Y -673.798,Z 1317.348,A 0.000,B 0.000,C 90.000,E1 98.681} C_DIS
LIN {X 0.158,Y -671.941,Z 1317.345,A 0.000,B 0.000,C 90.000,E1 98.163} C_DIS
LIN {X -0.171,Y -668.652,Z 1317.341,A 0.000,B 0.000,C 90.000,E1 97.466} C_DIS
LIN {X 0.225,Y -666.230,Z 1317.339,A 0.000,B 0.000,C 90.000,E1 96.947} C_DIS
LIN {X -0.152,Y -662.895,Z 1317.335,A 0.000,B 0.000,C 90.000,E1 96.372} C_DIS
LIN {X 0.107,Y -659.255,Z 1317.332,A 0.000,B 0.000,C 90.000,E1 95.739} C_DIS
LIN {X 0.232,Y -654.446,Z 1317.328,A 0.000,B 0.000,C 90.000,E1 94.992} C_DIS
LIN {X -0.231,Y -649.860,Z 1317.324,A 0.000,B 0.000,C 90.000,E1 94.416} C_DIS
LIN {X 0.085,Y -645.014,Z 1317.321,A 0.000,B 0.000,C 90.000,E1 93.784} C_DIS
LIN {X 0.064,Y -638.468,Z 1317.317,A 0.000,B 0.000,C 90.000,E1 93.037} C_DIS
LIN {X 0.080,Y -632.651,Z 1317.313,A 0.000,B 0.000,C 90.000,E1 92.407} C_DIS
LIN {X 0.172,Y -626.467,Z 1317.310,A 0.000,B 0.000,C 90.000,E1 91.776} C_DIS
LIN {X -0.061,Y -620.058,Z 1317.307,A 0.000,B 0.000,C 90.000,E1 91.203} C_DIS
LIN {X -0.085,Y -616.103,Z 1317.305,A 0.000,B 0.000,C 90.000,E1 90.859} C_DIS
LIN {X 0.151,Y -608.506,Z 1317.302,A 0.000,B 0.000,C 90.000,E1 90.286} C_DIS
LIN {X -0.299,Y -602.045,Z 1317.300,A 0.000,B 0.000,C 90.000,E1 89.943} C_DIS
LIN {X -0.282,Y -595.370,Z 1317.298,A 0.000,B 0.000,C 90.000,E1 89.599} C_DIS
LIN {X 0.143,Y -588.361,Z 1317.296,A 0.000,B 0.000,C 90.000,E1 89.255} C_DIS
LIN {X 0.076,Y -576.426,Z 1317.293,A 0.000,B 0.000,C 90.000,E1 88.797} C_DIS
LIN {X 0.236,Y -573.443,Z 1317.293,A 0.000,B 0.000,C 90.000,E1 88.625} C_DIS
LIN {X 0.027,Y -573.136,Z 1317.292,A 0.000,B 0.000,C 90.000,E1 88.625} C_DIS
LIN {X -0.065,Y -571.604,Z 1317.291,A 0.000,B 0.000,C 90.000,E1 88.453} C_DIS
LIN {X -0.108,Y -571.570,Z 1317.291,A 0.000,B 0.000,C 90.000,E1 88.453} C_DIS
LIN {X 0.278,Y -571.047,Z 1317.290,A 0.000,B 0.000,C 90.000,E1 88.108} C_DIS
LIN {X 0.193,Y -571.118,Z 1317.287,A 0.000,B 0.000,C 90.000,E1 87.707} C_DIS
LIN {X 0.046,Y -572.895,Z 1317.277,A 0.000,B 0.000,C 90.000,E1 85.812} C_DIS
LIN {X -0.256,Y -575.559,Z 1317.263,A 0.000,B 0.000,C 90.000,E1 83.394} C_DIS
LIN {X -0.192,Y -577.816,Z 1317.253,A 0.000,B 0.000,C 90.000,E1 81.489} C_DIS
LIN {X 0.226,Y -579.419,Z 1317.245,A 0.000,B 0.000,C 90.000,E1 80.095} C_DIS
LIN {X 0.100,Y -580.904,Z 1317.238,A 0.000,B 0.000,C 90.000,E1 78.757} C_DIS
LIN {X -0.121,Y -581.999,Z 1317.232,A 0.000,B 0.000,C 90.000,E1 77.701} C_DIS
LIN {X 0.242,Y -582.963,Z 1317.226,A 0.000,B 0.000,C 90.000,E1 76.589} C_DIS
LIN {X 0.092,Y -584.167,Z 1317.217,A 0.000,B 0.000,C 90.000,E1 74.991} C_DIS
LIN {X -0.272,Y -585.071,Z 1317.209,A 0.000,B 0.000,C 90.000,E1 73.685} C_DIS
LIN {X -0.127,Y -585.826,Z 1317.203,A 0.000,B 0.000,C 90.000,E1 72.598} C_DIS
LIN {X -0.208,Y -587.045,Z 1317.193,A 0.000,B 0.000,C 90.000,E1 70.732} C_DIS
LIN {X -0.204,Y -588.368,Z 1317.181,A 0.000,B 0.000,C 90.000,E1 68.592} C_DIS
LIN {X -0.039,Y -589.457,Z 1317.172,A 0.000,B 0.000,C 90.000,E1 66.975} C_DIS
LIN {X 0.042,Y -590.731,Z 1317.162,A 0.000,B 0.000,C 90.000,E1 65.101} C_DIS
LIN {X -0.240,Y -592.233,Z 1317.150,A 0.000,B 0.000,C 90.000,E1 62.999} C_DIS
LIN {X -0.026,Y -593.557,Z 1317.141,A 0.000,B 0.000,C 90.000,E1 61.385} C_DIS
LIN {X -0.124,Y -594.533,Z 1317.135,A 0.000,B 0.000,C 90.000,E1 60.333} C_DIS
LIN {X 0.001,Y -595.846,Z 1317.128,A 0.000,B 0.000,C 90.000,E1 58.997} C_DIS
LIN {X -0.228,Y -597.806,Z 1317.118,A 0.000,B 0.000,C 90.000,E1 57.168} C_DIS
LIN {X 0.275,Y -599.217,Z 1317.110,A 0.000,B 0.000,C 90.000,E1 55.801} C_DIS
LIN {X 0.057,Y -600.312,Z 1317.104,A 0.000,B 0.000,C 90.000,E1 54.769} C_DIS
LIN {X -0.036,Y -601.534,Z 1317.097,A 0.000,B 0.000,C 90.000,E1 53.463} C_DIS
LIN {X 0.013,Y -602.673,Z 1317.090,A 0.000,B 0.000,C 90.000,E1 52.145} C_DIS
LIN {X 0.081,Y -603.482,Z 1317.084,A 0.000,B 0.000,C 90.000,E1 51.090} C_DIS
LIN {X -0.168,Y -604.580,Z 1317.075,A 0.000,B 0.000,C 90.000,E1 49.542} C_DIS
LIN {X -0.320,Y -604.978,Z 1317.071,A 0.000,B 0.000,C 90.000,E1 48.771} C_DIS
LIN {X -0.214,Y -605.241,Z 1317.065,A 0.000,B 0.000,C 90.000,E1 47.715} C_DIS
LIN {X -0.285,Y -605.468,Z 1317.055,A 0.000,B 0.000,C 90.000,E1 45.891} C_DIS
LIN {X -0.009,Y -605.493,Z 1317.051,A 0.000,B 0.000,C 90.000,E1 45.081} C_DIS
LIN {X -0.120,Y -605.216,Z 1317.043,A 0.000,B 0.000,C 90.000,E1 43.785} C_DIS
LIN {X -0.001,Y -604.757,Z 1317.035,A 0.000,B 0.000,C 90.000,E1 42.204} C_DIS
LIN {X -0.102,Y -604.283,Z 1317.027,A 0.000,B 0.000,C 90.000,E1 40.906} C_DIS
LIN {X 0.247,Y -603.668,Z 1317.020,A 0.000,B 0.000,C 90.000,E1 39.564} C_DIS
LIN {X -0.046,Y -603.183,Z 1317.014,A 0.000,B 0.000,C 90.000,E1 38.543} C_DIS
LIN {X -0.344,Y -602.440,Z 1317.008,A 0.000,B 0.000,C 90.000,E1 37.523} C_DIS
LIN {X -0.065,Y -601.678,Z 1317.004,A 0.000,B 0.000,C 90.000,E1 36.710} C_DIS
LIN {X 0.079,Y -601.067,Z 1317.001,A 0.000,B 0.000,C 90.000,E1 36.171} C_DIS
LIN {X -0.020,Y -599.108,Z 1316.994,A 0.000,B 0.000,C 90.000,E1 34.865} C_DIS
LIN {X -0.348,Y -596.723,Z 1316.986,A 0.000,B 0.000,C 90.000,E1 33.579} C_DIS
LIN {X 0.002,Y -594.978,Z 1316.982,A 0.000,B 0.000,C 90.000,E1 32.752} C_DIS
LIN {X 0.223,Y -592.360,Z 1316.976,A 0.000,B 0.000,C 90.000,E1 31.671} C_DIS
LIN {X 0.211,Y -589.978,Z 1316.972,A 0.000,B 0.000,C 90.000,E1 30.875} C_DIS
LIN {X 0.291,Y -588.219,Z 1316.969,A 0.000,B 0.000,C 90.000,E1 30.335} C_DIS
LIN {X 0.235,Y -585.187,Z 1316.964,A 0.000,B 0.000,C 90.000,E1 29.539} C_DIS
LIN {X -0.008,Y -582.962,Z 1316.961,A 0.000,B 0.000,C 90.000,E1 29.027} C_DIS
LIN {X -0.185,Y -578.716,Z 1316.956,A 0.000,B 0.000,C 90.000,E1 28.103} C_DIS
LIN {X 0.237,Y -575.235,Z 1316.952,A 0.000,B 0.000,C 90.000,E1 27.385} C_DIS
LIN {X -0.070,Y -572.249,Z 1316.949,A 0.000,B 0.000,C 90.000,E1 26.873} C_DIS
LIN {X 0.031,Y -568.236,Z 1316.946,A 0.000,B 0.000,C 90.000,E1 26.181} C_DIS
LIN {X -0.073,Y -564.804,Z 1316.943,A 0.000,B 0.000,C 90.000,E1 25.643} C_DIS
LIN {X 0.156,Y -562.100,Z 1316.940,A 0.000,B 0.000,C 90.000,E1 25.207} C_DIS
LIN {X 0.269,Y -558.195,Z 1316.937,A 0.000,B 0.000,C 90.000,E1 24.643} C_DIS
LIN {X -0.078,Y -554.149,Z 1316.934,A 0.000,B 0.000,C 90.000,E1 24.131} C_DIS
LIN {X -0.138,Y -548.628,Z 1316.930,A 0.000,B 0.000,C 90.000,E1 23.439} C_DIS
LIN {X -0.210,Y -545.132,Z 1316.928,A 0.000,B 0.000,C 90.000,E1 23.025} C_DIS
LIN {X 0.050,Y -536.751,Z 1316.922,A 0.000,B 0.000,C 90.000,E1 22.025} C_DIS
LIN {X 0.110,Y -531.691,Z 1316.919,A 0.000,B 0.000,C 90.000,E1 21.461} C_DIS
LIN {X 0.251,Y -522.727,Z 1316.914,A 0.000,B 0.000,C 90.000,E1 20.482} C_DIS
LIN {X -0.005,Y -512.037,Z 1316.908,A 0.000,B 0.000,C 90.000,E1 19.396} C_DIS
LIN {X -0.104,Y -502.872,Z 1316.903,A 0.000,B 0.000,C 90.000,E1 18.471} C_DIS
LIN {X 0.066,Y -490.238,Z 1316.896,A 0.000,B 0.000,C 90.000,E1 17.221} C_DIS
LIN {X -0.031,Y -483.153,Z 1316.892,A 0.000,B 0.000,C 90.000,E1 16.551} C_DIS
LIN {X 0.074,Y -474.427,Z 1316.887,A 0.000,B 0.000,C 90.000,E1 15.733} C_DIS
LIN {X 0.220,Y -464.115,Z 1316.882,A 0.000,B 0.000,C 90.000,E1 14.773} C_DIS
LIN {X -0.026,Y -446.771,Z 1316.873,A 0.000,B 0.000,C 90.000,E1 13.175} C_DIS
LIN {X 0.151,Y -425.268,Z 1316.861,A 0.000,B 0.000,C 90.000,E1 10.950} C_DIS
LIN {X 0.078,Y -409.692,Z 1316.852,A 0.000,B 0.000,C 90.000,E1 9.265} C_DIS
LIN {X 0.017,Y -398.290,Z 1316.844,A 0.000,B 0.000,C 90.000,E1 7.992} C_DIS
LIN {X 0.126,Y -395.291,Z 1316.842,A 0.000,B 0.000,C 90.000,E1 7.530} C_DIS
LIN {X 0.089,Y -395.293,Z 1316.842,A 0.000,B 0.000,C 90.000,E1 7.530} C_DIS
LIN {X -0.062,Y -396.167,Z 1316.841,A 0.000,B 0.000,C 90.000,E1 7.409} C_DIS
LIN {X 0.160,Y -399.544,Z 1316.839,A 0.000,B 0.000,C 90.000,E1 7.068} C_DIS
LIN {X 0.028,Y -404.730,Z 1316.837,A 0.000,B 0.000,C 90.000,E1 6.720} C_DIS
LIN {X 0.194,Y -412.684,Z 1316.835,A 0.000,B 0.000,C 90.000,E1 6.201} C_DIS
LIN {X -0.039,Y -419.249,Z 1316.832,A 0.000,B 0.000,C 90.000,E1 5.796} C_DIS
LIN {X -0.042,Y -424.020,Z 1316.830,A 0.000,B 0.000,C 90.000,E1 5.454} C_DIS
LIN {X -0.222,Y -430.267,Z 1316.828,A 0.000,B 0.000,C 90.000,E1 4.992} C_DIS
LIN {X 0.081,Y -437.834,Z 1316.824,A 0.000,B 0.000,C 90.000,E1 4.302} C_DIS
LIN {X 0.094,Y -442.369,Z 1316.822,A 0.000,B 0.000,C 90.000,E1 3.898} C_DIS
LIN {X -0.167,Y -449.349,Z 1316.818,A 0.000,B 0.000,C 90.000,E1 3.269} C_DIS
LIN {X -0.160,Y -455.132,Z 1316.815,A 0.000,B 0.000,C 90.000,E1 2.694} C_DIS
LIN {X 0.212,Y -460.693,Z 1316.812,A 0.000,B 0.000,C 90.000,E1 2.064} C_DIS
LIN {X 0.127,Y -467.373,Z 1316.807,A 0.000,B 0.000,C 90.000,E1 1.318} C_DIS
LIN {X 0.164,Y -472.357,Z 1316.804,A 0.000,B 0.000,C 90.000,E1 0.688} C_DIS
LIN {X 0.069,Y -476.010,Z 1316.801,A 0.000,B 0.000,C 90.000,E1 0.229} C_DIS
LIN {X 0.125,Y -482.406,Z 1316.796,A 0.000,B 0.000,C 90.000,E1 359.312} C_DIS
LIN {X -0.092,Y -487.309,Z 1316.792,A 0.000,B 0.000,C 90.000,E1 358.568} C_DIS
LIN {X 0.241,Y -491.896,Z 1316.788,A 0.000,B 0.000,C 90.000,E1 357.764} C_DIS
LIN {X 0.106,Y -496.162,Z 1316.784,A 0.000,B 0.000,C 90.000,E1 357.020} C_DIS
LIN {X 0.034,Y -500.109,Z 1316.779,A 0.000,B 0.000,C 90.000,E1 356.274} C_DIS
LIN {X -0.001,Y -503.835,Z 1316.775,A 0.000,B 0.000,C 90.000,E1 355.527} C_DIS
LIN {X -0.197,Y -506.628,Z 1316.772,A 0.000,B 0.000,C 90.000,E1 354.951} C_DIS
LIN {X -0.022,Y -511.785,Z 1316.765,A 0.000,B 0.000,C 90.000,E1 353.742} C_DIS
LIN {X -0.163,Y -514.162,Z 1316.762,A 0.000,B 0.000,C 90.000,E1 353.166} C_DIS
LIN {X 0.196,Y -517.350,Z 1316.757,A 0.000,B 0.000,C 90.000,E1 352.243} C_DIS
LIN {X 0.077,Y -520.292,Z 1316.752,A 0.000,B 0.000,C 90.000,E1 351.376} C_DIS
LIN {X 0.068,Y -522.099,Z 1316.749,A 0.000,B 0.000,C 90.000,E1 350.792} C_DIS
LIN {X 0.008,Y -525.400,Z 1316.742,A 0.000,B 0.000,C 90.000,E1 349.634} C_DIS
LIN {X 0.062,Y -527.533,Z 1316.738,A 0.000,B 0.000,C 90.000,E1 348.757} C_DIS
LIN {X 0.140,Y -529.549,Z 1316.733,A 0.000,B 0.000,C 90.000,E1 347.881} C_DIS
LIN {X -0.161,Y -531.261,Z 1316.728,A 0.000,B 0.000,C 90.000,E1 347.048} C_DIS
LIN {X -0.043,Y -532.697,Z 1316.723,A 0.000,B 0.000,C 90.000,E1 346.172} C_DIS
LIN {X -0.256,Y -534.363,Z 1316.717,A 0.000,B 0.000,C 90.000,E1 345.046} C_DIS
LIN {X 0.022,Y -535.314,Z 1316.712,A 0.000,B 0.000,C 90.000,E1 344.157} C_DIS
LIN {X -0.207,Y -536.034,Z 1316.707,A 0.000,B 0.000,C 90.000,E1 343.323} C_DIS
LIN {X 0.038,Y -536.336,Z 1316.704,A 0.000,B 0.000,C 90.000,E1 342.725} C_DIS
LIN {X 0.021,Y -536.652,Z 1316.698,A 0.000,B 0.000,C 90.000,E1 341.583} C_DIS
LIN {X -0.030,Y -536.478,Z 1316.693,A 0.000,B 0.000,C 90.000,E1 340.732} C_DIS
LIN {X 0.129,Y -535.785,Z 1316.687,A 0.000,B 0.000,C 90.000,E1 339.571} C_DIS
LIN {X 0.067,Y -534.916,Z 1316.682,A 0.000,B 0.000,C 90.000,E1 338.720} C_DIS
LIN {X 0.191,Y -534.036,Z 1316.677,A 0.000,B 0.000,C 90.000,E1 337.847} C_DIS
LIN {X -0.099,Y -532.950,Z 1316.674,A 0.000,B 0.000,C 90.000,E1 337.305} C_DIS
LIN {X 0.100,Y -532.455,Z 1316.672,A 0.000,B 0.000,C 90.000,E1 336.997} C_DIS
LIN {X -0.291,Y -530.470,Z 1316.667,A 0.000,B 0.000,C 90.000,E1 336.177} C_DIS
LIN {X 0.003,Y -528.219,Z 1316.663,A 0.000,B 0.000,C 90.000,E1 335.281} C_DIS
LIN {X 0.053,Y -525.668,Z 1316.658,A 0.000,B 0.000,C 90.000,E1 334.409} C_DIS
LIN {X 0.046,Y -520.096,Z 1316.648,A 0.000,B 0.000,C 90.000,E1 332.666} C_DIS
LIN {X -0.107,Y -516.329,Z 1316.642,A 0.000,B 0.000,C 90.000,E1 331.513} C_DIS
LIN {X -0.071,Y -512.222,Z 1316.635,A 0.000,B 0.000,C 90.000,E1 330.333} C_DIS
LIN {X 0.159,Y -507.915,Z 1316.629,A 0.000,B 0.000,C 90.000,E1 329.125} C_DIS
LIN {X 0.058,Y -503.021,Z 1316.622,A 0.000,B 0.000,C 90.000,E1 327.946} C_DIS
LIN {X -0.011,Y -498.368,Z 1316.615,A 0.000,B 0.000,C 90.000,E1 326.755} C_DIS
LIN {X -0.132,Y -496.246,Z 1316.612,A 0.000,B 0.000,C 90.000,E1 326.167} C_DIS
LIN {X 0.002,Y -494.424,Z 1316.609,A 0.000,B 0.000,C 90.000,E1 325.548} C_DIS
LIN {X 0.208,Y -490.566,Z 1316.599,A 0.000,B 0.000,C 90.000,E1 323.703} C_DIS
LIN {X -0.101,Y -489.066,Z 1316.595,A 0.000,B 0.000,C 90.000,E1 323.130} C_DIS
LIN {X -0.259,Y -488.185,Z 1316.594,A 0.000,B 0.000,C 90.000,E1 322.844} C_DIS
LIN {X 0.265,Y -487.123,Z 1316.592,A 0.000,B 0.000,C 90.000,E1 322.477} C_DIS
LIN {X 0.101,Y -485.696,Z 1316.590,A 0.000,B 0.000,C 90.000,E1 322.190} C_DIS
LIN {X -0.133,Y -484.624,Z 1316.589,A 0.000,B 0.000,C 90.000,E1 322.065} C_DIS
LIN {X 0.132,Y -460.274,Z 1316.576,A 0.000,B 0.000,C 90.000,E1 319.666} C_DIS
LIN {X 0.181,Y -439.740,Z 1316.563,A 0.000,B 0.000,C 90.000,E1 317.391} C_DIS
LIN {X -0.046,Y -421.340,Z 1316.551,A 0.000,B 0.000,C 90.000,E1 315.121} C_DIS
LIN {X 0.229,Y -404.410,Z 1316.537,A 0.000,B 0.000,C 90.000,E1 312.690} C_DIS
LIN {X 0.077,Y -389.052,Z 1316.524,A 0.000,B 0.000,C 90.000,E1 310.253} C_DIS
LIN {X -0.022,Y -385.701,Z 1316.521,A 0.000,B 0.000,C 90.000,E1 309.688} C_DIS
LIN {X 0.238,Y -385.684,Z 1316.521,A 0.000,B 0.000,C 90.000,E1 309.644} C_DIS
LIN {X -0.118,Y -391.084,Z 1316.493,A 0.000,B 0.000,C 90.000,E1 304.739} C_DIS
LIN {X 0.121,Y -391.639,Z 1316.489,A 0.000,B 0.000,C 90.000,E1 303.992} C_DIS
LIN {X 0.019,Y -396.807,Z 1316.459,A 0.000,B 0.000,C 90.000,E1 298.693} C_DIS
LIN {X -0.111,Y -397.113,Z 1316.458,A 0.000,B 0.000,C 90.000,E1 298.359} C_DIS
LIN {X 0.045,Y -401.586,Z 1316.426,A 0.000,B 0.000,C 90.000,E1 292.717} C_DIS
LIN {X -0.065,Y -404.646,Z 1316.395,A 0.000,B 0.000,C 90.000,E1 287.149} C_DIS
LIN {X 0.021,Y -404.735,Z 1316.391,A 0.000,B 0.000,C 90.000,E1 286.441} C_DIS
LIN {X -0.083,Y -406.091,Z 1316.364,A 0.000,B 0.000,C 90.000,E1 281.591} C_DIS
LIN {X -0.076,Y -406.100,Z 1316.362,A 0.000,B 0.000,C 90.000,E1 281.243} C_DIS
LIN {X -0.039,Y -405.676,Z 1316.333,A 0.000,B 0.000,C 90.000,E1 276.030} C_DIS
LIN {X -0.031,Y -405.293,Z 1316.330,A 0.000,B 0.000,C 90.000,E1 275.334} C_DIS
LIN {X 0.039,Y -403.505,Z 1316.305,A 0.000,B 0.000,C 90.000,E1 270.802} C_DIS
LIN {X 0.007,Y -403.297,Z 1316.303,A 0.000,B 0.000,C 90.000,E1 270.458} C_DIS
LIN {X 0.191,Y -398.945,Z 1316.271,A 0.000,B 0.000,C 90.000,E1 264.837} C_DIS
LIN {X 0.058,Y -393.120,Z 1316.242,A 0.000,B 0.000,C 90.000,E1 259.567} C_DIS
LIN {X 0.019,Y -392.850,Z 1316.240,A 0.000,B 0.000,C 90.000,E1 259.218} C_DIS
LIN {X 0.133,Y -386.008,Z 1316.212,A 0.000,B 0.000,C 90.000,E1 254.212} C_DIS
LIN {X 0.072,Y -385.281,Z 1316.208,A 0.000,B 0.000,C 90.000,E1 253.504} C_DIS
LIN {X 0.094,Y -384.794,Z 1316.206,A 0.000,B 0.000,C 90.000,E1 253.142} C_DIS
LIN {X -0.035,Y -377.991,Z 1316.182,A 0.000,B 0.000,C 90.000,E1 248.827} C_DIS
LIN {X 0.053,Y -376.250,Z 1316.174,A 0.000,B 0.000,C 90.000,E1 247.358} C_DIS
LIN {X 0.154,Y -374.973,Z 1316.170,A 0.000,B 0.000,C 90.000,E1 246.613} C_DIS
LIN {X -0.111,Y -368.438,Z 1316.148,A 0.000,B 0.000,C 90.000,E1 242.615} C_DIS
LIN {X 0.193,Y -366.075,Z 1316.138,A 0.000,B 0.000,C 90.000,E1 240.717} C_DIS
LIN {X 0.099,Y -359.218,Z 1316.115,A 0.000,B 0.000,C 90.000,E1 236.628} C_DIS
LIN {X 0.176,Y -358.490,Z 1316.112,A 0.000,B 0.000,C 90.000,E1 236.087} C_DIS
LIN {X 0.138,Y -358.488,Z 1316.112,A 0.000,B 0.000,C 90.000,E1 236.087} C_DIS
LIN {X -0.192,Y -370.726,Z 1316.097,A 0.000,B 0.000,C 90.000,E1 233.497} C_DIS
LIN {X 0.173,Y -384.191,Z 1316.083,A 0.000,B 0.000,C 90.000,E1 230.884} C_DIS
LIN {X 0.059,Y -399.100,Z 1316.069,A 0.000,B 0.000,C 90.000,E1 228.405} C_DIS
LIN {X 0.052,Y -415.559,Z 1316.056,A 0.000,B 0.000,C 90.000,E1 225.972} C_DIS
LIN {X -0.070,Y -433.680,Z 1316.042,A 0.000,B 0.000,C 90.000,E1 223.623} C_DIS
LIN {X 0.233,Y -443.220,Z 1316.036,A 0.000,B 0.000,C 90.000,E1 222.447} C_DIS
LIN {X -0.035,Y -444.317,Z 1316.035,A 0.000,B 0.000,C 90.000,E1 222.324} C_DIS
LIN {X -0.003,Y -445.054,Z 1316.034,A 0.000,B 0.000,C 90.000,E1 222.162} C_DIS
LIN {X -0.025,Y -446.136,Z 1316.032,A 0.000,B 0.000,C 90.000,E1 221.838} C_DIS
LIN {X -0.044,Y -446.898,Z 1316.031,A 0.000,B 0.000,C 90.000,E1 221.515} C_DIS
LIN {X -0.033,Y -447.980,Z 1316.027,A 0.000,B 0.000,C 90.000,E1 220.862} C_DIS
LIN {X -0.014,Y -449.065,Z 1316.022,A 0.000,B 0.000,C 90.000,E1 219.886} C_DIS
LIN {X 0.002,Y -450.021,Z 1316.014,A 0.000,B 0.000,C 90.000,E1 218.588} C_DIS
LIN {X 0.222,Y -451.803,Z 1316.002,A 0.000,B 0.000,C 90.000,E1 216.297} C_DIS
LIN {X 0.035,Y -454.449,Z 1315.986,A 0.000,B 0.000,C 90.000,E1 213.420} C_DIS
LIN {X 0.049,Y -455.834,Z 1315.979,A 0.000,B 0.000,C 90.000,E1 212.133} C_DIS
LIN {X -0.096,Y -458.765,Z 1315.964,A 0.000,B 0.000,C 90.000,E1 209.589} C_DIS
LIN {X 0.051,Y -460.821,Z 1315.955,A 0.000,B 0.000,C 90.000,E1 207.975} C_DIS
LIN {X -0.125,Y -463.999,Z 1315.943,A 0.000,B 0.000,C 90.000,E1 205.771} C_DIS
LIN {X -0.212,Y -465.878,Z 1315.936,A 0.000,B 0.000,C 90.000,E1 204.515} C_DIS
LIN {X 0.105,Y -468.108,Z 1315.927,A 0.000,B 0.000,C 90.000,E1 202.898} C_DIS
LIN {X -0.048,Y -469.466,Z 1315.922,A 0.000,B 0.000,C 90.000,E1 201.972} C_DIS
LIN {X 0.051,Y -472.881,Z 1315.908,A 0.000,B 0.000,C 90.000,E1 199.450} C_DIS
LIN {X -0.011,Y -475.481,Z 1315.898,A 0.000,B 0.000,C 90.000,E1 197.583} C_DIS
LIN {X 0.012,Y -477.678,Z 1315.889,A 0.000,B 0.000,C 90.000,E1 196.024} C_DIS
LIN {X 0.096,Y -479.334,Z 1315.882,A 0.000,B 0.000,C 90.000,E1 194.773} C_DIS
LIN {X -0.059,Y -481.467,Z 1315.874,A 0.000,B 0.000,C 90.000,E1 193.244} C_DIS
LIN {X 0.168,Y -483.932,Z 1315.863,A 0.000,B 0.000,C 90.000,E1 191.366} C_DIS
LIN {X 0.002,Y -486.005,Z 1315.855,A 0.000,B 0.000,C 90.000,E1 189.849} C_DIS
LIN {X 0.033,Y -488.848,Z 1315.843,A 0.000,B 0.000,C 90.000,E1 187.701} C_DIS
LIN {X -0.022,Y -490.346,Z 1315.836,A 0.000,B 0.000,C 90.000,E1 186.486} C_DIS
LIN {X 0.215,Y -492.162,Z 1315.828,A 0.000,B 0.000,C 90.000,E1 184.935} C_DIS
LIN {X 0.154,Y -493.351,Z 1315.821,A 0.000,B 0.000,C 90.000,E1 183.726} C_DIS
LIN {X 0.077,Y -494.539,Z 1315.814,A 0.000,B 0.000,C 90.000,E1 182.522} C_DIS
LIN {X 0.014,Y -495.550,Z 1315.807,A 0.000,B 0.000,C 90.000,E1 181.318} C_DIS
LIN {X -0.181,Y -496.511,Z 1315.799,A 0.000,B 0.000,C 90.000,E1 179.828} C_DIS
LIN {X -0.092,Y -496.875,Z 1315.794,A 0.000,B 0.000,C 90.000,E1 178.912} C_DIS
LIN {X -0.121,Y -497.261,Z 1315.787,A 0.000,B 0.000,C 90.000,E1 177.707} C_DIS
LIN {X -0.141,Y -497.260,Z 1315.781,A 0.000,B 0.000,C 90.000,E1 176.502} C_DIS
LIN {X 0.114,Y -497.195,Z 1315.777,A 0.000,B 0.000,C 90.000,E1 175.869} C_DIS
LIN {X 0.228,Y -496.840,Z 1315.772,A 0.000,B 0.000,C 90.000,E1 174.951} C_DIS
LIN {X 0.235,Y -496.078,Z 1315.765,A 0.000,B 0.000,C 90.000,E1 173.742} C_DIS
LIN {X -0.267,Y -495.060,Z 1315.759,A 0.000,B 0.000,C 90.000,E1 172.591} C_DIS
LIN {X -0.064,Y -493.916,Z 1315.754,A 0.000,B 0.000,C 90.000,E1 171.659} C_DIS
LIN {X 0.057,Y -492.490,Z 1315.749,A 0.000,B 0.000,C 90.000,E1 170.735} C_DIS
LIN {X -0.144,Y -491.332,Z 1315.745,A 0.000,B 0.000,C 90.000,E1 170.151} C_DIS
LIN {X 0.027,Y -489.463,Z 1315.740,A 0.000,B 0.000,C 90.000,E1 169.218} C_DIS
LIN {X -0.080,Y -488.761,Z 1315.739,A 0.000,B 0.000,C 90.000,E1 168.926} C_DIS
LIN {X -0.060,Y -485.420,Z 1315.732,A 0.000,B 0.000,C 90.000,E1 167.701} C_DIS
LIN {X -0.182,Y -484.534,Z 1315.730,A 0.000,B 0.000,C 90.000,E1 167.409} C_DIS
LIN {X -0.127,Y -480.030,Z 1315.723,A 0.000,B 0.000,C 90.000,E1 166.172} C_DIS
LIN {X 0.006,Y -475.546,Z 1315.718,A 0.000,B 0.000,C 90.000,E1 165.227} C_DIS
LIN {X -0.164,Y -466.485,Z 1315.709,A 0.000,B 0.000,C 90.000,E1 163.685} C_DIS
LIN {X -0.147,Y -459.286,Z 1315.702,A 0.000,B 0.000,C 90.000,E1 162.417} C_DIS
LIN {X -0.030,Y -455.984,Z 1315.699,A 0.000,B 0.000,C 90.000,E1 161.764} C_DIS
LIN {X 0.200,Y -453.267,Z 1315.695,A 0.000,B 0.000,C 90.000,E1 161.094} C_DIS
LIN {X 0.094,Y -452.056,Z 1315.693,A 0.000,B 0.000,C 90.000,E1 160.786} C_DIS
LIN {X 0.147,Y -450.125,Z 1315.690,A 0.000,B 0.000,C 90.000,E1 160.134} C_DIS
LIN {X 0.062,Y -449.784,Z 1315.685,A 0.000,B 0.000,C 90.000,E1 159.337} C_DIS
LIN {X -0.208,Y -450.050,Z 1315.684,A 0.000,B 0.000,C 90.000,E1 159.209} C_DIS
LIN {X -0.097,Y -450.483,Z 1315.684,A 0.000,B 0.000,C 90.000,E1 159.082} C_DIS
LIN {X 0.014,Y -451.526,Z 1315.683,A 0.000,B 0.000,C 90.000,E1 158.954} C_DIS
LIN {X -0.065,Y -453.959,Z 1315.681,A 0.000,B 0.000,C 90.000,E1 158.646} C_DIS
LIN {X 0.039,Y -454.230,Z 1315.681,A 0.000,B 0.000,C 90.000,E1 158.592} C_DIS
LIN {X -0.180,Y -459.929,Z 1315.678,A 0.000,B 0.000,C 90.000,E1 158.103} C_DIS
LIN {X 0.166,Y -474.302,Z 1315.672,A 0.000,B 0.000,C 90.000,E1 156.922} C_DIS
LIN {X -0.079,Y -480.168,Z 1315.669,A 0.000,B 0.000,C 90.000,E1 156.485} C_DIS
LIN {X -0.091,Y -489.212,Z 1315.665,A 0.000,B 0.000,C 90.000,E1 155.741} C_DIS
LIN {X -0.051,Y -496.157,Z 1315.662,A 0.000,B 0.000,C 90.000,E1 155.101} C_DIS
LIN {X 0.192,Y -502.920,Z 1315.658,A 0.000,B 0.000,C 90.000,E1 154.409} C_DIS
LIN {X -0.004,Y -505.699,Z 1315.656,A 0.000,B 0.000,C 90.000,E1 154.152} C_DIS
LIN {X 0.080,Y -512.113,Z 1315.652,A 0.000,B 0.000,C 90.000,E1 153.435} C_DIS
LIN {X 0.087,Y -515.897,Z 1315.650,A 0.000,B 0.000,C 90.000,E1 152.999} C_DIS
LIN {X 0.104,Y -520.548,Z 1315.647,A 0.000,B 0.000,C 90.000,E1 152.410} C_DIS
LIN {X -0.090,Y -524.647,Z 1315.644,A 0.000,B 0.000,C 90.000,E1 151.847} C_DIS
LIN {X -0.008,Y -528.322,Z 1315.640,A 0.000,B 0.000,C 90.000,E1 151.257} C_DIS
LIN {X 0.101,Y -531.338,Z 1315.637,A 0.000,B 0.000,C 90.000,E1 150.667} C_DIS
LIN {X -0.229,Y -533.757,Z 1315.634,A 0.000,B 0.000,C 90.000,E1 150.127} C_DIS
LIN {X -0.081,Y -535.863,Z 1315.631,A 0.000,B 0.000,C 90.000,E1 149.537} C_DIS
LIN {X -0.096,Y -536.784,Z 1315.629,A 0.000,B 0.000,C 90.000,E1 149.253} C_DIS
LIN {X 0.074,Y -538.367,Z 1315.626,A 0.000,B 0.000,C 90.000,E1 148.663} C_DIS
LIN {X 0.259,Y -540.319,Z 1315.621,A 0.000,B 0.000,C 90.000,E1 147.788} C_DIS
LIN {X 0.008,Y -541.872,Z 1315.616,A 0.000,B 0.000,C 90.000,E1 146.962} C_DIS
LIN {X -0.247,Y -542.750,Z 1315.613,A 0.000,B 0.000,C 90.000,E1 146.421} C_DIS
LIN {X 0.036,Y -544.519,Z 1315.605,A 0.000,B 0.000,C 90.000,E1 144.975} C_DIS
LIN {X -0.104,Y -546.118,Z 1315.598,A 0.000,B 0.000,C 90.000,E1 143.577} C_DIS
LIN {X -0.165,Y -546.696,Z 1315.595,A 0.000,B 0.000,C 90.000,E1 143.050} C_DIS
LIN {X -0.208,Y -546.713,Z 1315.595,A 0.000,B 0.000,C 90.000,E1 143.050} C_DIS
LIN {X 0.164,Y -547.627,Z 1315.594,A 0.000,B 0.000,C 90.000,E1 142.844} C_DIS
LIN {X 0.020,Y -548.162,Z 1315.593,A 0.000,B 0.000,C 90.000,E1 142.718} C_DIS
LIN {X -0.169,Y -548.550,Z 1315.592,A 0.000,B 0.000,C 90.000,E1 142.557} C_DIS
LIN {X -0.211,Y -548.591,Z 1315.592,A 0.000,B 0.000,C 90.000,E1 142.557} C_DIS
LIN {X 0.066,Y -549.708,Z 1315.591,A 0.000,B 0.000,C 90.000,E1 142.431} C_DIS
LIN {X -0.178,Y -551.460,Z 1315.590,A 0.000,B 0.000,C 90.000,E1 142.271} C_DIS
LIN {X 0.261,Y -558.244,Z 1315.589,A 0.000,B 0.000,C 90.000,E1 141.984} C_DIS
LIN {X 0.177,Y -563.582,Z 1315.588,A 0.000,B 0.000,C 90.000,E1 141.823} C_DIS
LIN {X -0.280,Y -569.794,Z 1315.587,A 0.000,B 0.000,C 90.000,E1 141.618} C_DIS
LIN {X -0.068,Y -575.712,Z 1315.585,A 0.000,B 0.000,C 90.000,E1 141.295} C_DIS
LIN {X -0.029,Y -581.691,Z 1315.583,A 0.000,B 0.000,C 90.000,E1 140.928} C_DIS
LIN {X 0.117,Y -587.384,Z 1315.581,A 0.000,B 0.000,C 90.000,E1 140.517} C_DIS
LIN {X -0.167,Y -592.730,Z 1315.578,A 0.000,B 0.000,C 90.000,E1 140.114} C_DIS
LIN {X 0.036,Y -597.838,Z 1315.576,A 0.000,B 0.000,C 90.000,E1 139.622} C_DIS
LIN {X -0.048,Y -601.525,Z 1315.574,A 0.000,B 0.000,C 90.000,E1 139.256} C_DIS
LIN {X -0.246,Y -609.239,Z 1315.569,A 0.000,B 0.000,C 90.000,E1 138.405} C_DIS
LIN {X 0.114,Y -614.848,Z 1315.565,A 0.000,B 0.000,C 90.000,E1 137.634} C_DIS
LIN {X 0.355,Y -617.679,Z 1315.563,A 0.000,B 0.000,C 90.000,E1 137.229} C_DIS
LIN {X 0.193,Y -620.411,Z 1315.561,A 0.000,B 0.000,C 90.000,E1 136.863} C_DIS
LIN {X -0.381,Y -627.107,Z 1315.555,A 0.000,B 0.000,C 90.000,E1 135.891} C_DIS
LIN {X -0.128,Y -629.312,Z 1315.553,A 0.000,B 0.000,C 90.000,E1 135.486} C_DIS
LIN {X 0.024,Y -633.351,Z 1315.549,A 0.000,B 0.000,C 90.000,E1 134.838} C_DIS
LIN {X -0.384,Y -639.203,Z 1315.544,A 0.000,B 0.000,C 90.000,E1 133.866} C_DIS
LIN {X -0.178,Y -643.417,Z 1315.539,A 0.000,B 0.000,C 90.000,E1 133.095} C_DIS
LIN {X -0.050,Y -650.238,Z 1315.532,A 0.000,B 0.000,C 90.000,E1 131.838} C_DIS
LIN {X 0.273,Y -654.337,Z 1315.528,A 0.000,B 0.000,C 90.000,E1 131.067} C_DIS
LIN {X 0.174,Y -659.524,Z 1315.523,A 0.000,B 0.000,C 90.000,E1 130.092} C_DIS
LIN {X 0.138,Y -664.343,Z 1315.517,A 0.000,B 0.000,C 90.000,E1 129.116} C_DIS
LIN {X 0.170,Y -667.679,Z 1315.513,A 0.000,B 0.000,C 90.000,E1 128.382} C_DIS
LIN {X 0.233,Y -670.910,Z 1315.509,A 0.000,B 0.000,C 90.000,E1 127.649} C_DIS
LIN {X 0.335,Y -672.896,Z 1315.507,A 0.000,B 0.000,C 90.000,E1 127.156} C_DIS
LIN {X 0.046,Y -675.616,Z 1315.503,A 0.000,B 0.000,C 90.000,E1 126.457} C_DIS
LIN {X -0.216,Y -678.876,Z 1315.497,A 0.000,B 0.000,C 90.000,E1 125.518} C_DIS
LIN {X 0.110,Y -681.145,Z 1315.493,A 0.000,B 0.000,C 90.000,E1 124.771} C_DIS
LIN {X -0.097,Y -683.836,Z 1315.488,A 0.000,B 0.000,C 90.000,E1 123.833} C_DIS
LIN {X 0.284,Y -685.611,Z 1315.484,A 0.000,B 0.000,C 90.000,E1 123.086} C_DIS
LIN {X 0.313,Y -687.577,Z 1315.479,A 0.000,B 0.000,C 90.000,E1 122.133} C_DIS
LIN {X 0.007,Y -689.327,Z 1315.473,A 0.000,B 0.000,C 90.000,E1 121.209} C_DIS
LIN {X 0.079,Y -690.778,Z 1315.468,A 0.000,B 0.000,C 90.000,E1 120.256} C_DIS
LIN {X 0.052,Y -692.314,Z 1315.462,A 0.000,B 0.000,C 90.000,E1 119.077} C_DIS
LIN {X 0.170,Y -692.906,Z 1315.458,A 0.000,B 0.000,C 90.000,E1 118.359} C_DIS
LIN {X -0.076,Y -693.324,Z 1315.452,A 0.000,B 0.000,C 90.000,E1 117.436} C_DIS
LIN {X -0.020,Y -693.466,Z 1315.447,A 0.000,B 0.000,C 90.000,E1 116.488} C_DIS
LIN {X -0.147,Y -693.388,Z 1315.445,A 0.000,B 0.000,C 90.000,E1 116.027} C_DIS
LIN {X 0.295,Y -692.935,Z 1315.441,A 0.000,B 0.000,C 90.000,E1 115.283} C_DIS
LIN {X -0.087,Y -692.740,Z 1315.439,A 0.000,B 0.000,C 90.000,E1 115.079} C_DIS
LIN {X 0.111,Y -692.083,Z 1315.437,A 0.000,B 0.000,C 90.000,E1 114.591} C_DIS
LIN {X -0.276,Y -691.616,Z 1315.435,A 0.000,B 0.000,C 90.000,E1 114.387} C_DIS
LIN {X -0.080,Y -690.227,Z 1315.433,A 0.000,B 0.000,C 90.000,E1 113.898} C_DIS
LIN {X 0.272,Y -688.403,Z 1315.431,A 0.000,B 0.000,C 90.000,E1 113.515} C_DIS
LIN {X -0.404,Y -687.101,Z 1315.429,A 0.000,B 0.000,C 90.000,E1 113.334} C_DIS
LIN {X -0.291,Y -686.266,Z 1315.429,A 0.000,B 0.000,C 90.000,E1 113.206} C_DIS
LIN {X 0.137,Y -682.401,Z 1315.427,A 0.000,B 0.000,C 90.000,E1 112.823} C_DIS
LIN {X 0.278,Y -679.707,Z 1315.426,A 0.000,B 0.000,C 90.000,E1 112.589} C_DIS
LIN {X -0.152,Y -677.361,Z 1315.425,A 0.000,B 0.000,C 90.000,E1 112.514} C_DIS
LIN {X 0.182,Y -673.366,Z 1315.424,A 0.000,B 0.000,C 90.000,E1 112.333} C_DIS
LIN {X 0.190,Y -668.985,Z 1315.423,A 0.000,B 0.000,C 90.000,E1 112.206} C_DIS
LIN {X -0.231,Y -665.521,Z 1315.423,A 0.000,B 0.000,C 90.000,E1 112.153} C_DIS
LIN {X -0.155,Y -660.822,Z 1315.423,A 0.000,B 0.000,C 90.000,E1 112.078} C_DIS
LIN {X -0.273,Y -655.835,Z 1315.422,A 0.000,B 0.000,C 90.000,E1 112.025} C_DIS
LIN {X -0.074,Y -649.592,Z 1315.422,A 0.000,B 0.000,C 90.000,E1 111.972} C_DIS
LIN {X 0.070,Y -644.780,Z 1315.422,A 0.000,B 0.000,C 90.000,E1 111.897} C_DIS
LIN {X 0.147,Y -642.934,Z 1315.422,A 0.000,B 0.000,C 90.000,E1 111.844} C_DIS
LIN {X -0.139,Y -642.184,Z 1315.421,A 0.000,B 0.000,C 90.000,E1 111.844} C_DIS
LIN {X -0.180,Y -642.163,Z 1315.421,A 0.000,B 0.000,C 90.000,E1 111.844} C_DIS
LIN {X 0.299,Y -643.220,Z 1315.420,A 0.000,B 0.000,C 90.000,E1 111.589} C_DIS
LIN {X 0.104,Y -651.083,Z 1315.415,A 0.000,B 0.000,C 90.000,E1 110.610} C_DIS
LIN {X -0.090,Y -656.145,Z 1315.411,A 0.000,B 0.000,C 90.000,E1 109.885} C_DIS
LIN {X -0.067,Y -659.786,Z 1315.407,A 0.000,B 0.000,C 90.000,E1 109.268} C_DIS
LIN {X -0.178,Y -663.434,Z 1315.403,A 0.000,B 0.000,C 90.000,E1 108.544} C_DIS
LIN {X -0.260,Y -666.587,Z 1315.399,A 0.000,B 0.000,C 90.000,E1 107.819} C_DIS
LIN {X -0.232,Y -668.496,Z 1315.396,A 0.000,B 0.000,C 90.000,E1 107.330} C_DIS
LIN {X 0.179,Y -670.976,Z 1315.392,A 0.000,B 0.000,C 90.000,E1 106.567} C_DIS
LIN {X 0.232,Y -672.474,Z 1315.390,A 0.000,B 0.000,C 90.000,E1 106.079} C_DIS
LIN {X 0.047,Y -674.321,Z 1315.385,A 0.000,B 0.000,C 90.000,E1 105.371} C_DIS
LIN {X -0.063,Y -675.409,Z 1315.383,A 0.000,B 0.000,C 90.000,E1 104.898} C_DIS
LIN {X -0.098,Y -677.163,Z 1315.377,A 0.000,B 0.000,C 90.000,E1 103.939} C_DIS
LIN {X -0.146,Y -677.558,Z 1315.376,A 0.000,B 0.000,C 90.000,E1 103.703} C_DIS
LIN {X 0.223,Y -678.269,Z 1315.372,A 0.000,B 0.000,C 90.000,E1 102.952} C_DIS
LIN {X 0.098,Y -678.694,Z 1315.368,A 0.000,B 0.000,C 90.000,E1 102.243} C_DIS
LIN {X 0.013,Y -678.760,Z 1315.365,A 0.000,B 0.000,C 90.000,E1 101.771} C_DIS
LIN {X -0.074,Y -678.626,Z 1315.363,A 0.000,B 0.000,C 90.000,E1 101.299} C_DIS
LIN {X 0.326,Y -678.051,Z 1315.359,A 0.000,B 0.000,C 90.000,E1 100.546} C_DIS
LIN {X 0.229,Y -677.395,Z 1315.356,A 0.000,B 0.000,C 90.000,E1 100.074} C_DIS
LIN {X 0.060,Y -677.028,Z 1315.355,A 0.000,B 0.000,C 90.000,E1 99.849} C_DIS
LIN {X -0.048,Y -675.968,Z 1315.352,A 0.000,B 0.000,C 90.000,E1 99.378} C_DIS
LIN {X -0.273,Y -674.577,Z 1315.349,A 0.000,B 0.000,C 90.000,E1 98.916} C_DIS
LIN {X 0.163,Y -672.909,Z 1315.347,A 0.000,B 0.000,C 90.000,E1 98.398} C_DIS
LIN {X 0.093,Y -671.984,Z 1315.345,A 0.000,B 0.000,C 90.000,E1 98.163} C_DIS
LIN {X -0.235,Y -668.658,Z 1315.341,A 0.000,B 0.000,C 90.000,E1 97.466} C_DIS
LIN {X 0.161,Y -666.228,Z 1315.339,A 0.000,B 0.000,C 90.000,E1 96.947} C_DIS
LIN {X -0.215,Y -662.863,Z 1315.335,A 0.000,B 0.000,C 90.000,E1 96.372} C_DIS
LIN {X 0.138,Y -659.978,Z 1315.333,A 0.000,B 0.000,C 90.000,E1 95.853} C_DIS
LIN {X -0.185,Y -656.801,Z 1315.330,A 0.000,B 0.000,C 90.000,E1 95.391} C_DIS
LIN {X 0.067,Y -653.440,Z 1315.327,A 0.000,B 0.000,C 90.000,E1 94.878} C_DIS
LIN {X -0.295,Y -649.747,Z 1315.324,A 0.000,B 0.000,C 90.000,E1 94.416} C_DIS
LIN {X -0.148,Y -644.705,Z 1315.321,A 0.000,B 0.000,C 90.000,E1 93.784} C_DIS
LIN {X -0.170,Y -638.105,Z 1315.317,A 0.000,B 0.000,C 90.000,E1 93.037} C_DIS
LIN {X -0.280,Y -631.079,Z 1315.313,A 0.000,B 0.000,C 90.000,E1 92.293} C_DIS
LIN {X -0.167,Y -624.772,Z 1315.309,A 0.000,B 0.000,C 90.000,E1 91.661} C_DIS
LIN {X -0.270,Y -616.973,Z 1315.305,A 0.000,B 0.000,C 90.000,E1 90.974} C_DIS
LIN {X -0.305,Y -615.531,Z 1315.305,A 0.000,B 0.000,C 90.000,E1 90.859} C_DIS
LIN {X 0.034,Y -609.654,Z 1315.302,A 0.000,B 0.000,C 90.000,E1 90.401} C_DIS
LIN {X 0.033,Y -603.105,Z 1315.300,A 0.000,B 0.000,C 90.000,E1 90.000} C_DIS
LIN {X -0.062,Y -596.421,Z 1315.298,A 0.000,B 0.000,C 90.000,E1 89.656} C_DIS
LIN {X -0.254,Y -589.612,Z 1315.296,A 0.000,B 0.000,C 90.000,E1 89.370} C_DIS
LIN {X 0.239,Y -576.153,Z 1315.293,A 0.000,B 0.000,C 90.000,E1 88.797} C_DIS
LIN {X -0.054,Y -573.247,Z 1315.293,A 0.000,B 0.000,C 90.000,E1 88.682} C_DIS
LIN {X -0.100,Y -573.160,Z 1315.293,A 0.000,B 0.000,C 90.000,E1 88.682} C_DIS
LIN {X 0.055,Y -571.398,Z 1315.292,A 0.000,B 0.000,C 90.000,E1 88.453} C_DIS
LIN {X 0.013,Y -571.387,Z 1315.292,A 0.000,B 0.000,C 90.000,E1 88.453} C_DIS
LIN {X -0.173,Y -570.853,Z 1315.290,A 0.000,B 0.000,C 90.000,E1 88.165} C_DIS
LIN {X -0.259,Y -570.957,Z 1315.287,A 0.000,B 0.000,C 90.000,E1 87.764} C_DIS
LIN {X -0.141,Y -572.201,Z 1315.280,A 0.000,B 0.000,C 90.000,E1 86.388} C_DIS
LIN {X -0.090,Y -574.476,Z 1315.268,A 0.000,B 0.000,C 90.000,E1 84.204} C_DIS
LIN {X 0.184,Y -576.020,Z 1315.260,A 0.000,B 0.000,C 90.000,E1 82.818} C_DIS
LIN {X 0.128,Y -577.994,Z 1315.251,A 0.000,B 0.000,C 90.000,E1 81.197} C_DIS
LIN {X -0.016,Y -579.600,Z 1315.244,A 0.000,B 0.000,C 90.000,E1 79.859} C_DIS
LIN {X -0.137,Y -581.043,Z 1315.236,A 0.000,B 0.000,C 90.000,E1 78.522} C_DIS
LIN {X -0.123,Y -582.348,Z 1315.229,A 0.000,B 0.000,C 90.000,E1 77.173} C_DIS
LIN {X -0.324,Y -583.238,Z 1315.223,A 0.000,B 0.000,C 90.000,E1 76.117} C_DIS
LIN {X 0.092,Y -584.418,Z 1315.214,A 0.000,B 0.000,C 90.000,E1 74.464} C_DIS
LIN {X 0.123,Y -585.482,Z 1315.205,A 0.000,B 0.000,C 90.000,E1 72.851} C_DIS
LIN {X -0.201,Y -586.503,Z 1315.196,A 0.000,B 0.000,C 90.000,E1 71.275} C_DIS
LIN {X -0.033,Y -587.183,Z 1315.190,A 0.000,B 0.000,C 90.000,E1 70.188} C_DIS
LIN {X 0.308,Y -588.413,Z 1315.180,A 0.000,B 0.000,C 90.000,E1 68.284} C_DIS
LIN {X 0.045,Y -589.326,Z 1315.172,A 0.000,B 0.000,C 90.000,E1 66.975} C_DIS
LIN {X 0.123,Y -590.602,Z 1315.162,A 0.000,B 0.000,C 90.000,E1 65.101} C_DIS
LIN {X -0.162,Y -592.091,Z 1315.150,A 0.000,B 0.000,C 90.000,E1 62.999} C_DIS
LIN {X 0.048,Y -593.441,Z 1315.141,A 0.000,B 0.000,C 90.000,E1 61.385} C_DIS
LIN {X -0.138,Y -595.494,Z 1315.129,A 0.000,B 0.000,C 90.000,E1 59.282} C_DIS
LIN {X -0.257,Y -597.992,Z 1315.116,A 0.000,B 0.000,C 90.000,E1 56.914} C_DIS
LIN {X -0.015,Y -599.678,Z 1315.107,A 0.000,B 0.000,C 90.000,E1 55.308} C_DIS
LIN {X 0.017,Y -600.941,Z 1315.100,A 0.000,B 0.000,C 90.000,E1 53.989} C_DIS
LIN {X -0.062,Y -602.122,Z 1315.093,A 0.000,B 0.000,C 90.000,E1 52.683} C_DIS
LIN {X -0.114,Y -603.183,Z 1315.085,A 0.000,B 0.000,C 90.000,E1 51.376} C_DIS
LIN {X -0.111,Y -604.451,Z 1315.075,A 0.000,B 0.000,C 90.000,E1 49.542} C_DIS
LIN {X -0.264,Y -604.854,Z 1315.071,A 0.000,B 0.000,C 90.000,E1 48.771} C_DIS
LIN {X -0.159,Y -605.131,Z 1315.065,A 0.000,B 0.000,C 90.000,E1 47.715} C_DIS
LIN {X -0.233,Y -605.358,Z 1315.055,A 0.000,B 0.000,C 90.000,E1 45.891} C_DIS
LIN {X 0.042,Y -605.385,Z 1315.051,A 0.000,B 0.000,C 90.000,E1 45.081} C_DIS
LIN {X -0.071,Y -605.150,Z 1315.043,A 0.000,B 0.000,C 90.000,E1 43.785} C_DIS
LIN {X 0.296,Y -604.607,Z 1315.033,A 0.000,B 0.000,C 90.000,E1 41.919} C_DIS
LIN {X 0.198,Y -604.105,Z 1315.026,A 0.000,B 0.000,C 90.000,E1 40.620} C_DIS
LIN {X -0.045,Y -603.384,Z 1315.017,A 0.000,B 0.000,C 90.000,E1 39.072} C_DIS
LIN {X 0.035,Y -602.756,Z 1315.011,A 0.000,B 0.000,C 90.000,E1 38.016} C_DIS
LIN {X -0.047,Y -602.075,Z 1315.007,A 0.000,B 0.000,C 90.000,E1 37.237} C_DIS
LIN {X -0.131,Y -601.255,Z 1315.003,A 0.000,B 0.000,C 90.000,E1 36.457} C_DIS
LIN {X -0.117,Y -600.569,Z 1315.000,A 0.000,B 0.000,C 90.000,E1 35.931} C_DIS
LIN {X -0.323,Y -599.034,Z 1314.994,A 0.000,B 0.000,C 90.000,E1 34.898} C_DIS
LIN {X -0.311,Y -596.644,Z 1314.986,A 0.000,B 0.000,C 90.000,E1 33.579} C_DIS
LIN {X -0.063,Y -594.291,Z 1314.981,A 0.000,B 0.000,C 90.000,E1 32.498} C_DIS
LIN {X 0.260,Y -592.314,Z 1314.976,A 0.000,B 0.000,C 90.000,E1 31.671} C_DIS
LIN {X -0.260,Y -589.918,Z 1314.972,A 0.000,B 0.000,C 90.000,E1 30.924} C_DIS
LIN {X -0.183,Y -588.172,Z 1314.969,A 0.000,B 0.000,C 90.000,E1 30.384} C_DIS
LIN {X 0.270,Y -585.144,Z 1314.964,A 0.000,B 0.000,C 90.000,E1 29.539} C_DIS
LIN {X 0.026,Y -582.920,Z 1314.961,A 0.000,B 0.000,C 90.000,E1 29.027} C_DIS
LIN {X -0.152,Y -578.674,Z 1314.956,A 0.000,B 0.000,C 90.000,E1 28.103} C_DIS
LIN {X 0.269,Y -575.193,Z 1314.952,A 0.000,B 0.000,C 90.000,E1 27.385} C_DIS
LIN {X -0.038,Y -572.208,Z 1314.949,A 0.000,B 0.000,C 90.000,E1 26.873} C_DIS
LIN {X 0.062,Y -568.196,Z 1314.946,A 0.000,B 0.000,C 90.000,E1 26.181} C_DIS
LIN {X -0.043,Y -564.760,Z 1314.943,A 0.000,B 0.000,C 90.000,E1 25.643} C_DIS
LIN {X 0.089,Y -561.091,Z 1314.939,A 0.000,B 0.000,C 90.000,E1 25.079} C_DIS
LIN {X 0.299,Y -558.146,Z 1314.937,A 0.000,B 0.000,C 90.000,E1 24.643} C_DIS
LIN {X -0.017,Y -554.088,Z 1314.934,A 0.000,B 0.000,C 90.000,E1 24.131} C_DIS
LIN {X -0.079,Y -548.572,Z 1314.930,A 0.000,B 0.000,C 90.000,E1 23.439} C_DIS
LIN {X -0.151,Y -545.078,Z 1314.928,A 0.000,B 0.000,C 90.000,E1 23.025} C_DIS
LIN {X -0.005,Y -536.563,Z 1314.922,A 0.000,B 0.000,C 90.000,E1 22.025} C_DIS
LIN {X -0.029,Y -531.387,Z 1314.919,A 0.000,B 0.000,C 90.000,E1 21.461} C_DIS
LIN {X 0.089,Y -522.397,Z 1314.914,A 0.000,B 0.000,C 90.000,E1 20.482} C_DIS
LIN {X 0.014,Y -511.913,Z 1314.908,A 0.000,B 0.000,C 90.000,E1 19.396} C_DIS
LIN {X -0.077,Y -502.724,Z 1314.903,A 0.000,B 0.000,C 90.000,E1 18.471} C_DIS
LIN {X 0.166,Y -488.865,Z 1314.895,A 0.000,B 0.000,C 90.000,E1 17.094} C_DIS
LIN {X 0.107,Y -483.124,Z 1314.892,A 0.000,B 0.000,C 90.000,E1 16.551} C_DIS
LIN {X -0.178,Y -474.487,Z 1314.888,A 0.000,B 0.000,C 90.000,E1 15.788} C_DIS
LIN {X -0.034,Y -464.118,Z 1314.882,A 0.000,B 0.000,C 90.000,E1 14.828} C_DIS
LIN {X 0.142,Y -443.733,Z 1314.872,A 0.000,B 0.000,C 90.000,E1 12.883} C_DIS
LIN {X -0.166,Y -425.093,Z 1314.861,A 0.000,B 0.000,C 90.000,E1 11.007} C_DIS
LIN {X -0.146,Y -408.135,Z 1314.851,A 0.000,B 0.000,C 90.000,E1 9.151} C_DIS
LIN {X -0.019,Y -398.457,Z 1314.845,A 0.000,B 0.000,C 90.000,E1 8.049} C_DIS
LIN {X -0.026,Y -395.395,Z 1314.842,A 0.000,B 0.000,C 90.000,E1 7.587} C_DIS
LIN {X -0.061,Y -395.385,Z 1314.842,A 0.000,B 0.000,C 90.000,E1 7.587} C_DIS
LIN {X 0.046,Y -395.959,Z 1314.842,A 0.000,B 0.000,C 90.000,E1 7.466} C_DIS
LIN {X -0.166,Y -399.854,Z 1314.839,A 0.000,B 0.000,C 90.000,E1 7.125} C_DIS
LIN {X -0.209,Y -405.821,Z 1314.837,A 0.000,B 0.000,C 90.000,E1 6.720} C_DIS
LIN {X -0.091,Y -412.099,Z 1314.835,A 0.000,B 0.000,C 90.000,E1 6.315} C_DIS
LIN {X 0.105,Y -418.643,Z 1314.833,A 0.000,B 0.000,C 90.000,E1 5.853} C_DIS
LIN {X 0.111,Y -421.977,Z 1314.831,A 0.000,B 0.000,C 90.000,E1 5.625} C_DIS
LIN {X 0.039,Y -429.686,Z 1314.828,A 0.000,B 0.000,C 90.000,E1 5.049} C_DIS
LIN {X -0.037,Y -437.280,Z 1314.825,A 0.000,B 0.000,C 90.000,E1 4.416} C_DIS
LIN {X -0.166,Y -443.308,Z 1314.822,A 0.000,B 0.000,C 90.000,E1 3.898} C_DIS
LIN {X -0.045,Y -449.230,Z 1314.818,A 0.000,B 0.000,C 90.000,E1 3.326} C_DIS
LIN {X -0.014,Y -455.020,Z 1314.815,A 0.000,B 0.000,C 90.000,E1 2.751} C_DIS
LIN {X -0.091,Y -460.673,Z 1314.812,A 0.000,B 0.000,C 90.000,E1 2.178} C_DIS
LIN {X -0.091,Y -467.336,Z 1314.808,A 0.000,B 0.000,C 90.000,E1 1.432} C_DIS
LIN {X 0.096,Y -473.554,Z 1314.804,A 0.000,B 0.000,C 90.000,E1 0.630} C_DIS
LIN {X 0.010,Y -477.179,Z 1314.801,A 0.000,B 0.000,C 90.000,E1 0.172} C_DIS
LIN {X 0.130,Y -483.108,Z 1314.796,A 0.000,B 0.000,C 90.000,E1 359.312} C_DIS
LIN {X -0.082,Y -488.007,Z 1314.792,A 0.000,B 0.000,C 90.000,E1 358.568} C_DIS
LIN {X -0.233,Y -492.594,Z 1314.788,A 0.000,B 0.000,C 90.000,E1 357.822} C_DIS
LIN {X 0.130,Y -496.872,Z 1314.784,A 0.000,B 0.000,C 90.000,E1 357.020} C_DIS
LIN {X 0.066,Y -500.833,Z 1314.779,A 0.000,B 0.000,C 90.000,E1 356.274} C_DIS
LIN {X 0.038,Y -504.556,Z 1314.775,A 0.000,B 0.000,C 90.000,E1 355.527} C_DIS
LIN {X -0.154,Y -507.335,Z 1314.772,A 0.000,B 0.000,C 90.000,E1 354.951} C_DIS
LIN {X 0.033,Y -512.527,Z 1314.765,A 0.000,B 0.000,C 90.000,E1 353.742} C_DIS
LIN {X -0.103,Y -514.912,Z 1314.762,A 0.000,B 0.000,C 90.000,E1 353.166} C_DIS
LIN {X -0.247,Y -518.126,Z 1314.757,A 0.000,B 0.000,C 90.000,E1 352.299} C_DIS
LIN {X 0.156,Y -521.067,Z 1314.752,A 0.000,B 0.000,C 90.000,E1 351.376} C_DIS
LIN {X 0.153,Y -522.870,Z 1314.749,A 0.000,B 0.000,C 90.000,E1 350.792} C_DIS
LIN {X 0.104,Y -526.182,Z 1314.743,A 0.000,B 0.000,C 90.000,E1 349.634} C_DIS
LIN {X 0.168,Y -528.365,Z 1314.738,A 0.000,B 0.000,C 90.000,E1 348.757} C_DIS
LIN {X -0.229,Y -530.993,Z 1314.731,A 0.000,B 0.000,C 90.000,E1 347.645} C_DIS
LIN {X 0.005,Y -532.627,Z 1314.726,A 0.000,B 0.000,C 90.000,E1 346.756} C_DIS
LIN {X 0.136,Y -534.025,Z 1314.722,A 0.000,B 0.000,C 90.000,E1 345.880} C_DIS
LIN {X -0.109,Y -535.258,Z 1314.717,A 0.000,B 0.000,C 90.000,E1 345.046} C_DIS
LIN {X 0.130,Y -535.950,Z 1314.714,A 0.000,B 0.000,C 90.000,E1 344.448} C_DIS
LIN {X -0.089,Y -536.729,Z 1314.709,A 0.000,B 0.000,C 90.000,E1 343.614} C_DIS
LIN {X 0.212,Y -537.300,Z 1314.704,A 0.000,B 0.000,C 90.000,E1 342.725} C_DIS
LIN {X 0.210,Y -537.597,Z 1314.698,A 0.000,B 0.000,C 90.000,E1 341.583} C_DIS
LIN {X 0.167,Y -537.443,Z 1314.693,A 0.000,B 0.000,C 90.000,E1 340.732} C_DIS
LIN {X -0.089,Y -537.171,Z 1314.690,A 0.000,B 0.000,C 90.000,E1 340.188} C_DIS
LIN {X -0.136,Y -536.539,Z 1314.685,A 0.000,B 0.000,C 90.000,E1 339.337} C_DIS
LIN {X 0.215,Y -535.323,Z 1314.679,A 0.000,B 0.000,C 90.000,E1 338.156} C_DIS
LIN {X -0.072,Y -535.006,Z 1314.677,A 0.000,B 0.000,C 90.000,E1 337.901} C_DIS
LIN {X -0.065,Y -534.550,Z 1314.676,A 0.000,B 0.000,C 90.000,E1 337.614} C_DIS
LIN {X 0.141,Y -533.904,Z 1314.674,A 0.000,B 0.000,C 90.000,E1 337.305} C_DIS
LIN {X -0.147,Y -533.445,Z 1314.672,A 0.000,B 0.000,C 90.000,E1 337.050} C_DIS
LIN {X 0.054,Y -532.757,Z 1314.671,A 0.000,B 0.000,C 90.000,E1 336.741} C_DIS
LIN {X -0.236,Y -532.242,Z 1314.669,A 0.000,B 0.000,C 90.000,E1 336.485} C_DIS
LIN {X -0.140,Y -530.125,Z 1314.664,A 0.000,B 0.000,C 90.000,E1 335.613} C_DIS
LIN {X 0.153,Y -527.674,Z 1314.660,A 0.000,B 0.000,C 90.000,E1 334.717} C_DIS
LIN {X -0.045,Y -522.123,Z 1314.650,A 0.000,B 0.000,C 90.000,E1 332.999} C_DIS
LIN {X 0.203,Y -517.413,Z 1314.642,A 0.000,B 0.000,C 90.000,E1 331.513} C_DIS
LIN {X 0.252,Y -513.286,Z 1314.635,A 0.000,B 0.000,C 90.000,E1 330.333} C_DIS
LIN {X -0.203,Y -508.864,Z 1314.629,A 0.000,B 0.000,C 90.000,E1 329.203} C_DIS
LIN {X -0.024,Y -503.937,Z 1314.622,A 0.000,B 0.000,C 90.000,E1 327.995} C_DIS
LIN {X 0.072,Y -499.127,Z 1314.616,A 0.000,B 0.000,C 90.000,E1 326.786} C_DIS
LIN {X 0.094,Y -496.004,Z 1314.611,A 0.000,B 0.000,C 90.000,E1 325.881} C_DIS
LIN {X -0.180,Y -494.313,Z 1314.607,A 0.000,B 0.000,C 90.000,E1 325.308} C_DIS
LIN {X -0.105,Y -492.709,Z 1314.602,A 0.000,B 0.000,C 90.000,E1 324.402} C_DIS
LIN {X -0.001,Y -491.841,Z 1314.599,A 0.000,B 0.000,C 90.000,E1 323.783} C_DIS
LIN {X 0.230,Y -490.301,Z 1314.594,A 0.000,B 0.000,C 90.000,E1 322.844} C_DIS
LIN {X -0.081,Y -489.071,Z 1314.590,A 0.000,B 0.000,C 90.000,E1 322.271} C_DIS
LIN {X -0.240,Y -488.313,Z 1314.589,A 0.000,B 0.000,C 90.000,E1 321.984} C_DIS
LIN {X -0.099,Y -487.393,Z 1314.587,A 0.000,B 0.000,C 90.000,E1 321.662} C_DIS
LIN {X 0.119,Y -486.241,Z 1314.585,A 0.000,B 0.000,C 90.000,E1 321.331} C_DIS
LIN {X 0.186,Y -485.445,Z 1314.584,A 0.000,B 0.000,C 90.000,E1 321.170} C_DIS
LIN {X -0.050,Y -484.262,Z 1314.584,A 0.000,B 0.000,C 90.000,E1 321.045} C_DIS
LIN {X -0.235,Y -462.883,Z 1314.572,A 0.000,B 0.000,C 90.000,E1 318.933} C_DIS
LIN {X -0.042,Y -442.607,Z 1314.559,A 0.000,B 0.000,C 90.000,E1 316.620} C_DIS
LIN {X 0.251,Y -423.319,Z 1314.545,A 0.000,B 0.000,C 90.000,E1 314.109} C_DIS
LIN {X -0.071,Y -405.815,Z 1314.531,A 0.000,B 0.000,C 90.000,E1 311.595} C_DIS
LIN {X 0.124,Y -391.038,Z 1314.517,A 0.000,B 0.000,C 90.000,E1 309.116} C_DIS
LIN {X -0.030,Y -386.834,Z 1314.513,A 0.000,B 0.000,C 90.000,E1 308.382} C_DIS
LIN {X -0.067,Y -386.805,Z 1314.513,A 0.000,B 0.000,C 90.000,E1 308.382} C_DIS
LIN {X 0.055,Y -391.345,Z 1314.492,A 0.000,B 0.000,C 90.000,E1 304.485} C_DIS
LIN {X -0.122,Y -397.056,Z 1314.458,A 0.000,B 0.000,C 90.000,E1 298.487} C_DIS
LIN {X 0.183,Y -401.447,Z 1314.427,A 0.000,B 0.000,C 90.000,E1 292.823} C_DIS
LIN {X -0.107,Y -401.676,Z 1314.425,A 0.000,B 0.000,C 90.000,E1 292.514} C_DIS
LIN {X -0.076,Y -404.536,Z 1314.396,A 0.000,B 0.000,C 90.000,E1 287.275} C_DIS
LIN {X 0.024,Y -404.763,Z 1314.394,A 0.000,B 0.000,C 90.000,E1 286.913} C_DIS
LIN {X -0.070,Y -406.151,Z 1314.363,A 0.000,B 0.000,C 90.000,E1 281.366} C_DIS
LIN {X 0.035,Y -405.647,Z 1314.334,A 0.000,B 0.000,C 90.000,E1 276.144} C_DIS
LIN {X 0.040,Y -405.627,Z 1314.332,A 0.000,B 0.000,C 90.000,E1 275.796} C_DIS
LIN {X 0.112,Y -403.554,Z 1314.305,A 0.000,B 0.000,C 90.000,E1 270.917} C_DIS
LIN {X 0.047,Y -403.078,Z 1314.301,A 0.000,B 0.000,C 90.000,E1 270.229} C_DIS
LIN {X -0.126,Y -399.026,Z 1314.272,A 0.000,B 0.000,C 90.000,E1 265.008} C_DIS
LIN {X 0.188,Y -398.153,Z 1314.268,A 0.000,B 0.000,C 90.000,E1 264.261} C_DIS
LIN {X 0.045,Y -392.949,Z 1314.241,A 0.000,B 0.000,C 90.000,E1 259.342} C_DIS
LIN {X 0.003,Y -392.514,Z 1314.239,A 0.000,B 0.000,C 90.000,E1 258.993} C_DIS
LIN {X 0.151,Y -386.146,Z 1314.213,A 0.000,B 0.000,C 90.000,E1 254.338} C_DIS
LIN {X 0.111,Y -385.026,Z 1314.207,A 0.000,B 0.000,C 90.000,E1 253.268} C_DIS
LIN {X -0.017,Y -378.160,Z 1314.183,A 0.000,B 0.000,C 90.000,E1 248.954} C_DIS
LIN {X 0.196,Y -375.923,Z 1314.173,A 0.000,B 0.000,C 90.000,E1 247.102} C_DIS
LIN {X -0.184,Y -369.134,Z 1314.151,A 0.000,B 0.000,C 90.000,E1 243.127} C_DIS
LIN {X 0.045,Y -366.285,Z 1314.138,A 0.000,B 0.000,C 90.000,E1 240.873} C_DIS
LIN {X -0.062,Y -360.460,Z 1314.120,A 0.000,B 0.000,C 90.000,E1 237.502} C_DIS
LIN {X -0.099,Y -360.472,Z 1314.119,A 0.000,B 0.000,C 90.000,E1 237.502} C_DIS
LIN {X -0.204,Y -372.656,Z 1314.104,A 0.000,B 0.000,C 90.000,E1 234.769} C_DIS
LIN {X -0.017,Y -385.529,Z 1314.090,A 0.000,B 0.000,C 90.000,E1 232.190} C_DIS
LIN {X -0.053,Y -399.786,Z 1314.076,A 0.000,B 0.000,C 90.000,E1 229.703} C_DIS
LIN {X 0.253,Y -415.522,Z 1314.063,A 0.000,B 0.000,C 90.000,E1 227.229} C_DIS
LIN {X -0.177,Y -432.849,Z 1314.049,A 0.000,B 0.000,C 90.000,E1 224.919} C_DIS
LIN {X -0.042,Y -443.477,Z 1314.042,A 0.000,B 0.000,C 90.000,E1 223.581} C_DIS
LIN {X -0.041,Y -444.645,Z 1314.041,A 0.000,B 0.000,C 90.000,E1 223.419} C_DIS
LIN {X -0.052,Y -445.415,Z 1314.040,A 0.000,B 0.000,C 90.000,E1 223.257} C_DIS
LIN {X -0.063,Y -446.004,Z 1314.039,A 0.000,B 0.000,C 90.000,E1 223.095} C_DIS
LIN {X -0.078,Y -446.902,Z 1314.038,A 0.000,B 0.000,C 90.000,E1 222.771} C_DIS
LIN {X -0.091,Y -447.582,Z 1314.036,A 0.000,B 0.000,C 90.000,E1 222.447} C_DIS
LIN {X 0.221,Y -448.565,Z 1314.032,A 0.000,B 0.000,C 90.000,E1 221.757} C_DIS
LIN {X -0.098,Y -449.396,Z 1314.027,A 0.000,B 0.000,C 90.000,E1 220.825} C_DIS
LIN {X -0.027,Y -450.240,Z 1314.018,A 0.000,B 0.000,C 90.000,E1 219.197} C_DIS
LIN {X -0.094,Y -452.416,Z 1314.002,A 0.000,B 0.000,C 90.000,E1 216.297} C_DIS
LIN {X 0.021,Y -454.734,Z 1313.987,A 0.000,B 0.000,C 90.000,E1 213.706} C_DIS
LIN {X 0.149,Y -456.430,Z 1313.978,A 0.000,B 0.000,C 90.000,E1 212.084} C_DIS
LIN {X 0.033,Y -459.372,Z 1313.964,A 0.000,B 0.000,C 90.000,E1 209.539} C_DIS
LIN {X -0.208,Y -461.437,Z 1313.955,A 0.000,B 0.000,C 90.000,E1 207.975} C_DIS
LIN {X 0.050,Y -464.620,Z 1313.943,A 0.000,B 0.000,C 90.000,E1 205.720} C_DIS
LIN {X -0.023,Y -466.489,Z 1313.936,A 0.000,B 0.000,C 90.000,E1 204.463} C_DIS
LIN {X -0.012,Y -467.858,Z 1313.931,A 0.000,B 0.000,C 90.000,E1 203.515} C_DIS
LIN {X -0.091,Y -470.062,Z 1313.922,A 0.000,B 0.000,C 90.000,E1 201.950} C_DIS
LIN {X -0.112,Y -473.049,Z 1313.910,A 0.000,B 0.000,C 90.000,E1 199.758} C_DIS
LIN {X -0.022,Y -475.743,Z 1313.899,A 0.000,B 0.000,C 90.000,E1 197.873} C_DIS
LIN {X -0.163,Y -478.376,Z 1313.889,A 0.000,B 0.000,C 90.000,E1 196.024} C_DIS
LIN {X -0.069,Y -480.108,Z 1313.882,A 0.000,B 0.000,C 90.000,E1 194.773} C_DIS
LIN {X -0.100,Y -482.268,Z 1313.874,A 0.000,B 0.000,C 90.000,E1 193.231} C_DIS
LIN {X 0.035,Y -484.781,Z 1313.863,A 0.000,B 0.000,C 90.000,E1 191.366} C_DIS
LIN {X -0.116,Y -486.881,Z 1313.855,A 0.000,B 0.000,C 90.000,E1 189.849} C_DIS
LIN {X 0.056,Y -489.361,Z 1313.844,A 0.000,B 0.000,C 90.000,E1 187.992} C_DIS
LIN {X -0.102,Y -491.335,Z 1313.836,A 0.000,B 0.000,C 90.000,E1 186.486} C_DIS
LIN {X 0.153,Y -493.196,Z 1313.828,A 0.000,B 0.000,C 90.000,E1 184.935} C_DIS
LIN {X -0.040,Y -494.816,Z 1313.819,A 0.000,B 0.000,C 90.000,E1 183.440} C_DIS
LIN {X 0.048,Y -495.721,Z 1313.814,A 0.000,B 0.000,C 90.000,E1 182.522} C_DIS
LIN {X 0.003,Y -496.786,Z 1313.807,A 0.000,B 0.000,C 90.000,E1 181.318} C_DIS
LIN {X -0.170,Y -497.848,Z 1313.799,A 0.000,B 0.000,C 90.000,E1 179.828} C_DIS
LIN {X -0.197,Y -498.372,Z 1313.792,A 0.000,B 0.000,C 90.000,E1 178.625} C_DIS
LIN {X -0.074,Y -498.728,Z 1313.787,A 0.000,B 0.000,C 90.000,E1 177.707} C_DIS
LIN {X -0.204,Y -498.814,Z 1313.779,A 0.000,B 0.000,C 90.000,E1 176.216} C_DIS
LIN {X -0.168,Y -498.602,Z 1313.772,A 0.000,B 0.000,C 90.000,E1 175.008} C_DIS
LIN {X 0.215,Y -497.782,Z 1313.764,A 0.000,B 0.000,C 90.000,E1 173.457} C_DIS
LIN {X -0.114,Y -497.102,Z 1313.759,A 0.000,B 0.000,C 90.000,E1 172.591} C_DIS
LIN {X 0.201,Y -496.432,Z 1313.755,A 0.000,B 0.000,C 90.000,E1 171.951} C_DIS
LIN {X 0.164,Y -494.234,Z 1313.747,A 0.000,B 0.000,C 90.000,E1 170.443} C_DIS
LIN {X -0.118,Y -492.477,Z 1313.742,A 0.000,B 0.000,C 90.000,E1 169.567} C_DIS
LIN {X 0.169,Y -491.217,Z 1313.739,A 0.000,B 0.000,C 90.000,E1 168.926} C_DIS
LIN {X -0.037,Y -489.777,Z 1313.735,A 0.000,B 0.000,C 90.000,E1 168.342} C_DIS
LIN {X -0.005,Y -486.406,Z 1313.729,A 0.000,B 0.000,C 90.000,E1 167.117} C_DIS
LIN {X -0.125,Y -485.470,Z 1313.727,A 0.000,B 0.000,C 90.000,E1 166.825} C_DIS
LIN {X -0.060,Y -480.902,Z 1313.720,A 0.000,B 0.000,C 90.000,E1 165.589} C_DIS
LIN {X 0.204,Y -476.512,Z 1313.715,A 0.000,B 0.000,C 90.000,E1 164.629} C_DIS
LIN {X 0.238,Y -469.478,Z 1313.708,A 0.000,B 0.000,C 90.000,E1 163.378} C_DIS
LIN {X -0.174,Y -460.016,Z 1313.698,A 0.000,B 0.000,C 90.000,E1 161.692} C_DIS
LIN {X -0.226,Y -457.793,Z 1313.696,A 0.000,B 0.000,C 90.000,E1 161.221} C_DIS
LIN {X 0.021,Y -455.347,Z 1313.692,A 0.000,B 0.000,C 90.000,E1 160.550} C_DIS
LIN {X -0.075,Y -454.338,Z 1313.690,A 0.000,B 0.000,C 90.000,E1 160.242} C_DIS
LIN {X -0.115,Y -453.103,Z 1313.686,A 0.000,B 0.000,C 90.000,E1 159.444} C_DIS
LIN {X 0.058,Y -453.665,Z 1313.683,A 0.000,B 0.000,C 90.000,E1 158.954} C_DIS
LIN {X 0.018,Y -453.686,Z 1313.683,A 0.000,B 0.000,C 90.000,E1 158.954} C_DIS
LIN {X 0.098,Y -454.583,Z 1313.682,A 0.000,B 0.000,C 90.000,E1 158.773} C_DIS
LIN {X -0.109,Y -455.655,Z 1313.681,A 0.000,B 0.000,C 90.000,E1 158.518} C_DIS
LIN {X 0.275,Y -455.703,Z 1313.681,A 0.000,B 0.000,C 90.000,E1 158.465} C_DIS
LIN {X 0.157,Y -457.684,Z 1313.680,A 0.000,B 0.000,C 90.000,E1 158.284} C_DIS
LIN {X 0.031,Y -458.901,Z 1313.679,A 0.000,B 0.000,C 90.000,E1 158.156} C_DIS
LIN {X 0.258,Y -462.171,Z 1313.677,A 0.000,B 0.000,C 90.000,E1 157.847} C_DIS
LIN {X 0.156,Y -478.693,Z 1313.670,A 0.000,B 0.000,C 90.000,E1 156.538} C_DIS
LIN {X -0.072,Y -489.049,Z 1313.665,A 0.000,B 0.000,C 90.000,E1 155.717} C_DIS
LIN {X 0.156,Y -494.825,Z 1313.662,A 0.000,B 0.000,C 90.000,E1 155.177} C_DIS
LIN {X -0.057,Y -501.653,Z 1313.659,A 0.000,B 0.000,C 90.000,E1 154.537} C_DIS
LIN {X 0.124,Y -505.785,Z 1313.656,A 0.000,B 0.000,C 90.000,E1 154.101} C_DIS
LIN {X 0.208,Y -512.230,Z 1313.652,A 0.000,B 0.000,C 90.000,E1 153.384} C_DIS
LIN {X -0.254,Y -515.998,Z 1313.650,A 0.000,B 0.000,C 90.000,E1 152.999} C_DIS
LIN {X -0.070,Y -519.562,Z 1313.647,A 0.000,B 0.000,C 90.000,E1 152.538} C_DIS
LIN {X -0.024,Y -523.751,Z 1313.644,A 0.000,B 0.000,C 90.000,E1 151.948} C_DIS
LIN {X -0.198,Y -527.516,Z 1313.641,A 0.000,B 0.000,C 90.000,E1 151.385} C_DIS
LIN {X -0.247,Y -531.342,Z 1313.637,A 0.000,B 0.000,C 90.000,E1 150.667} C_DIS
LIN {X -0.117,Y -533.783,Z 1313.634,A 0.000,B 0.000,C 90.000,E1 150.078} C_DIS
LIN {X -0.141,Y -534.858,Z 1313.632,A 0.000,B 0.000,C 90.000,E1 149.793} C_DIS
LIN {X 0.014,Y -536.698,Z 1313.629,A 0.000,B 0.000,C 90.000,E1 149.203} C_DIS
LIN {X 0.181,Y -538.284,Z 1313.626,A 0.000,B 0.000,C 90.000,E1 148.614} C_DIS
LIN {X -0.097,Y -540.181,Z 1313.621,A 0.000,B 0.000,C 90.000,E1 147.788} C_DIS
LIN {X 0.105,Y -541.716,Z 1313.616,A 0.000,B 0.000,C 90.000,E1 146.914} C_DIS
LIN {X -0.133,Y -542.915,Z 1313.612,A 0.000,B 0.000,C 90.000,E1 146.087} C_DIS
LIN {X -0.328,Y -544.340,Z 1313.605,A 0.000,B 0.000,C 90.000,E1 144.975} C_DIS
LIN {X -0.290,Y -546.264,Z 1313.597,A 0.000,B 0.000,C 90.000,E1 143.417} C_DIS
LIN {X -0.106,Y -546.547,Z 1313.596,A 0.000,B 0.000,C 90.000,E1 143.256} C_DIS
LIN {X -0.078,Y -548.628,Z 1313.594,A 0.000,B 0.000,C 90.000,E1 142.970} C_DIS
LIN {X 0.065,Y -551.633,Z 1313.593,A 0.000,B 0.000,C 90.000,E1 142.798} C_DIS
LIN {X -0.276,Y -559.638,Z 1313.592,A 0.000,B 0.000,C 90.000,E1 142.557} C_DIS
LIN {X 0.068,Y -566.300,Z 1313.590,A 0.000,B 0.000,C 90.000,E1 142.271} C_DIS
LIN {X 0.101,Y -572.510,Z 1313.589,A 0.000,B 0.000,C 90.000,E1 141.984} C_DIS
LIN {X -0.091,Y -578.170,Z 1313.587,A 0.000,B 0.000,C 90.000,E1 141.662} C_DIS
LIN {X 0.027,Y -581.366,Z 1313.586,A 0.000,B 0.000,C 90.000,E1 141.457} C_DIS
LIN {X -0.059,Y -585.651,Z 1313.584,A 0.000,B 0.000,C 90.000,E1 141.170} C_DIS
LIN {X -0.072,Y -589.956,Z 1313.583,A 0.000,B 0.000,C 90.000,E1 140.848} C_DIS
LIN {X -0.126,Y -593.906,Z 1313.581,A 0.000,B 0.000,C 90.000,E1 140.517} C_DIS
LIN {X 0.293,Y -599.000,Z 1313.578,A 0.000,B 0.000,C 90.000,E1 139.989} C_DIS
LIN {X 0.127,Y -602.645,Z 1313.576,A 0.000,B 0.000,C 90.000,E1 139.622} C_DIS
LIN {X 0.200,Y -607.185,Z 1313.573,A 0.000,B 0.000,C 90.000,E1 139.094} C_DIS
LIN {X -0.090,Y -611.464,Z 1313.570,A 0.000,B 0.000,C 90.000,E1 138.609} C_DIS
LIN {X -0.221,Y -618.043,Z 1313.565,A 0.000,B 0.000,C 90.000,E1 137.715} C_DIS
LIN {X -0.023,Y -620.710,Z 1313.563,A 0.000,B 0.000,C 90.000,E1 137.310} C_DIS
LIN {X -0.269,Y -628.847,Z 1313.556,A 0.000,B 0.000,C 90.000,E1 136.053} C_DIS
LIN {X 0.005,Y -636.890,Z 1313.548,A 0.000,B 0.000,C 90.000,E1 134.636} C_DIS
LIN {X 0.068,Y -643.184,Z 1313.542,A 0.000,B 0.000,C 90.000,E1 133.500} C_DIS
LIN {X 0.147,Y -650.534,Z 1313.534,A 0.000,B 0.000,C 90.000,E1 132.123} C_DIS
LIN {X -0.006,Y -655.801,Z 1313.529,A 0.000,B 0.000,C 90.000,E1 131.148} C_DIS
LIN {X -0.111,Y -660.170,Z 1313.524,A 0.000,B 0.000,C 90.000,E1 130.297} C_DIS
LIN {X -0.147,Y -664.857,Z 1313.518,A 0.000,B 0.000,C 90.000,E1 129.322} C_DIS
LIN {X -0.023,Y -669.150,Z 1313.513,A 0.000,B 0.000,C 90.000,E1 128.338} C_DIS
LIN {X 0.051,Y -673.151,Z 1313.508,A 0.000,B 0.000,C 90.000,E1 127.363} C_DIS
LIN {X 0.301,Y -676.692,Z 1313.502,A 0.000,B 0.000,C 90.000,E1 126.377} C_DIS
LIN {X 0.051,Y -679.043,Z 1313.498,A 0.000,B 0.000,C 90.000,E1 125.678} C_DIS
LIN {X 0.213,Y -681.301,Z 1313.494,A 0.000,B 0.000,C 90.000,E1 124.945} C_DIS
LIN {X 0.002,Y -683.334,Z 1313.490,A 0.000,B 0.000,C 90.000,E1 124.246} C_DIS
LIN {X -0.001,Y -685.748,Z 1313.485,A 0.000,B 0.000,C 90.000,E1 123.293} C_DIS
LIN {X 0.031,Y -687.775,Z 1313.480,A 0.000,B 0.000,C 90.000,E1 122.339} C_DIS
LIN {X 0.085,Y -689.513,Z 1313.474,A 0.000,B 0.000,C 90.000,E1 121.386} C_DIS
LIN {X -0.196,Y -691.025,Z 1313.469,A 0.000,B 0.000,C 90.000,E1 120.463} C_DIS
LIN {X -0.217,Y -692.601,Z 1313.463,A 0.000,B 0.000,C 90.000,E1 119.283} C_DIS
LIN {X -0.094,Y -693.316,Z 1313.459,A 0.000,B 0.000,C 90.000,E1 118.565} C_DIS
LIN {X -0.330,Y -693.795,Z 1313.453,A 0.000,B 0.000,C 90.000,E1 117.641} C_DIS
LIN {X 0.047,Y -694.044,Z 1313.448,A 0.000,B 0.000,C 90.000,E1 116.668} C_DIS
LIN {X -0.385,Y -694.038,Z 1313.446,A 0.000,B 0.000,C 90.000,E1 116.232} C_DIS
LIN {X 0.364,Y -693.709,Z 1313.442,A 0.000,B 0.000,C 90.000,E1 115.463} C_DIS
LIN {X -0.062,Y -693.278,Z 1313.439,A 0.000,B 0.000,C 90.000,E1 115.027} C_DIS
LIN {X 0.430,Y -692.593,Z 1313.436,A 0.000,B 0.000,C 90.000,E1 114.515} C_DIS
LIN {X -0.243,Y -692.069,Z 1313.435,A 0.000,B 0.000,C 90.000,E1 114.335} C_DIS
LIN {X 0.239,Y -690.635,Z 1313.432,A 0.000,B 0.000,C 90.000,E1 113.823} C_DIS
LIN {X -0.203,Y -688.072,Z 1313.430,A 0.000,B 0.000,C 90.000,E1 113.387} C_DIS
LIN {X -0.089,Y -687.398,Z 1313.429,A 0.000,B 0.000,C 90.000,E1 113.259} C_DIS
LIN {X 0.023,Y -686.469,Z 1313.429,A 0.000,B 0.000,C 90.000,E1 113.131} C_DIS
LIN {X 0.262,Y -680.306,Z 1313.426,A 0.000,B 0.000,C 90.000,E1 112.589} C_DIS
LIN {X -0.165,Y -678.100,Z 1313.425,A 0.000,B 0.000,C 90.000,E1 112.514} C_DIS
LIN {X 0.086,Y -673.943,Z 1313.424,A 0.000,B 0.000,C 90.000,E1 112.333} C_DIS
LIN {X 0.158,Y -667.346,Z 1313.423,A 0.000,B 0.000,C 90.000,E1 112.153} C_DIS
LIN {X -0.385,Y -665.334,Z 1313.423,A 0.000,B 0.000,C 90.000,E1 112.153} C_DIS
LIN {X 0.139,Y -659.301,Z 1313.422,A 0.000,B 0.000,C 90.000,E1 112.025} C_DIS
LIN {X 0.226,Y -654.522,Z 1313.422,A 0.000,B 0.000,C 90.000,E1 111.972} C_DIS
LIN {X 0.031,Y -650.023,Z 1313.422,A 0.000,B 0.000,C 90.000,E1 111.972} C_DIS
LIN {X 0.101,Y -644.673,Z 1313.422,A 0.000,B 0.000,C 90.000,E1 111.897} C_DIS
LIN {X 0.091,Y -642.722,Z 1313.422,A 0.000,B 0.000,C 90.000,E1 111.844} C_DIS
LIN {X -0.114,Y -642.186,Z 1313.421,A 0.000,B 0.000,C 90.000,E1 111.844} C_DIS
LIN {X -0.155,Y -642.128,Z 1313.421,A 0.000,B 0.000,C 90.000,E1 111.844} C_DIS
LIN {X 0.240,Y -643.227,Z 1313.420,A 0.000,B 0.000,C 90.000,E1 111.589} C_DIS
LIN {X 0.043,Y -651.032,Z 1313.415,A 0.000,B 0.000,C 90.000,E1 110.610} C_DIS
LIN {X -0.152,Y -656.101,Z 1313.410,A 0.000,B 0.000,C 90.000,E1 109.885} C_DIS
LIN {X -0.130,Y -659.736,Z 1313.407,A 0.000,B 0.000,C 90.000,E1 109.268} C_DIS
LIN {X -0.242,Y -663.381,Z 1313.403,A 0.000,B 0.000,C 90.000,E1 108.544} C_DIS
LIN {X -0.324,Y -666.554,Z 1313.399,A 0.000,B 0.000,C 90.000,E1 107.819} C_DIS
LIN {X 0.342,Y -668.488,Z 1313.396,A 0.000,B 0.000,C 90.000,E1 107.275} C_DIS
LIN {X 0.114,Y -670.962,Z 1313.392,A 0.000,B 0.000,C 90.000,E1 106.567} C_DIS
LIN {X 0.167,Y -672.436,Z 1313.389,A 0.000,B 0.000,C 90.000,E1 106.079} C_DIS
LIN {X -0.018,Y -674.275,Z 1313.385,A 0.000,B 0.000,C 90.000,E1 105.371} C_DIS
LIN {X -0.129,Y -675.365,Z 1313.383,A 0.000,B 0.000,C 90.000,E1 104.898} C_DIS
LIN {X -0.164,Y -677.115,Z 1313.377,A 0.000,B 0.000,C 90.000,E1 103.939} C_DIS
LIN {X -0.213,Y -677.503,Z 1313.376,A 0.000,B 0.000,C 90.000,E1 103.703} C_DIS
LIN {X 0.308,Y -678.183,Z 1313.372,A 0.000,B 0.000,C 90.000,E1 102.939} C_DIS
LIN {X 0.030,Y -678.642,Z 1313.368,A 0.000,B 0.000,C 90.000,E1 102.243} C_DIS
LIN {X -0.056,Y -678.728,Z 1313.365,A 0.000,B 0.000,C 90.000,E1 101.771} C_DIS
LIN {X -0.143,Y -678.591,Z 1313.363,A 0.000,B 0.000,C 90.000,E1 101.299} C_DIS
LIN {X 0.257,Y -678.019,Z 1313.359,A 0.000,B 0.000,C 90.000,E1 100.546} C_DIS
LIN {X 0.159,Y -677.386,Z 1313.356,A 0.000,B 0.000,C 90.000,E1 100.074} C_DIS
LIN {X -0.009,Y -677.019,Z 1313.355,A 0.000,B 0.000,C 90.000,E1 99.849} C_DIS
LIN {X -0.117,Y -675.976,Z 1313.352,A 0.000,B 0.000,C 90.000,E1 99.378} C_DIS
LIN {X 0.325,Y -674.591,Z 1313.349,A 0.000,B 0.000,C 90.000,E1 98.859} C_DIS
LIN {X 0.094,Y -672.919,Z 1313.347,A 0.000,B 0.000,C 90.000,E1 98.398} C_DIS
LIN {X 0.024,Y -672.025,Z 1313.345,A 0.000,B 0.000,C 90.000,E1 98.163} C_DIS
LIN {X 0.360,Y -668.662,Z 1313.341,A 0.000,B 0.000,C 90.000,E1 97.409} C_DIS
LIN {X 0.093,Y -666.225,Z 1313.339,A 0.000,B 0.000,C 90.000,E1 96.947} C_DIS
LIN {X 0.284,Y -662.132,Z 1313.335,A 0.000,B 0.000,C 90.000,E1 96.201} C_DIS
LIN {X -0.024,Y -659.133,Z 1313.332,A 0.000,B 0.000,C 90.000,E1 95.739} C_DIS
LIN {X 0.202,Y -655.058,Z 1313.328,A 0.000,B 0.000,C 90.000,E1 95.106} C_DIS
LIN {X -0.152,Y -651.500,Z 1313.326,A 0.000,B 0.000,C 90.000,E1 94.645} C_DIS
LIN {X 0.179,Y -648.611,Z 1313.324,A 0.000,B 0.000,C 90.000,E1 94.245} C_DIS
LIN {X -0.216,Y -644.507,Z 1313.321,A 0.000,B 0.000,C 90.000,E1 93.784} C_DIS
LIN {X -0.155,Y -638.991,Z 1313.318,A 0.000,B 0.000,C 90.000,E1 93.154} C_DIS
LIN {X -0.102,Y -633.182,Z 1313.314,A 0.000,B 0.000,C 90.000,E1 92.522} C_DIS
LIN {X 0.148,Y -629.534,Z 1313.312,A 0.000,B 0.000,C 90.000,E1 92.121} C_DIS
LIN {X -0.239,Y -624.505,Z 1313.309,A 0.000,B 0.000,C 90.000,E1 91.661} C_DIS
LIN {X 0.121,Y -616.463,Z 1313.305,A 0.000,B 0.000,C 90.000,E1 90.917} C_DIS
LIN {X -0.164,Y -609.015,Z 1313.302,A 0.000,B 0.000,C 90.000,E1 90.401} C_DIS
LIN {X -0.126,Y -602.419,Z 1313.300,A 0.000,B 0.000,C 90.000,E1 90.000} C_DIS
LIN {X -0.234,Y -595.651,Z 1313.298,A 0.000,B 0.000,C 90.000,E1 89.656} C_DIS
LIN {X 0.040,Y -588.348,Z 1313.296,A 0.000,B 0.000,C 90.000,E1 89.312} C_DIS
LIN {X 0.057,Y -577.775,Z 1313.294,A 0.000,B 0.000,C 90.000,E1 88.912} C_DIS
LIN {X 0.202,Y -573.087,Z 1313.293,A 0.000,B 0.000,C 90.000,E1 88.682} C_DIS
LIN {X 0.164,Y -573.012,Z 1313.293,A 0.000,B 0.000,C 90.000,E1 88.682} C_DIS
LIN {X 0.097,Y -571.096,Z 1313.292,A 0.000,B 0.000,C 90.000,E1 88.453} C_DIS
LIN {X 0.055,Y -571.084,Z 1313.292,A 0.000,B 0.000,C 90.000,E1 88.453} C_DIS
LIN {X 0.225,Y -570.662,Z 1313.290,A 0.000,B 0.000,C 90.000,E1 88.108} C_DIS
LIN {X -0.148,Y -570.807,Z 1313.287,A 0.000,B 0.000,C 90.000,E1 87.707} C_DIS
LIN {X 0.242,Y -571.631,Z 1313.283,A 0.000,B 0.000,C 90.000,E1 86.849} C_DIS
LIN {X 0.013,Y -574.423,Z 1313.268,A 0.000,B 0.000,C 90.000,E1 84.147} C_DIS
LIN {X -0.084,Y -576.257,Z 1313.259,A 0.000,B 0.000,C 90.000,E1 82.527} C_DIS
LIN {X 0.225,Y -577.937,Z 1313.251,A 0.000,B 0.000,C 90.000,E1 81.141} C_DIS
LIN {X 0.078,Y -579.545,Z 1313.243,A 0.000,B 0.000,C 90.000,E1 79.803} C_DIS
LIN {X -0.047,Y -580.971,Z 1313.236,A 0.000,B 0.000,C 90.000,E1 78.465} C_DIS
LIN {X 0.195,Y -582.508,Z 1313.227,A 0.000,B 0.000,C 90.000,E1 76.825} C_DIS
LIN {X -0.198,Y -583.533,Z 1313.219,A 0.000,B 0.000,C 90.000,E1 75.519} C_DIS
LIN {X 0.326,Y -584.324,Z 1313.214,A 0.000,B 0.000,C 90.000,E1 74.393} C_DIS
LIN {X -0.036,Y -585.182,Z 1313.206,A 0.000,B 0.000,C 90.000,E1 73.087} C_DIS
LIN {X 0.192,Y -586.218,Z 1313.197,A 0.000,B 0.000,C 90.000,E1 71.456} C_DIS
LIN {X 0.024,Y -587.086,Z 1313.190,A 0.000,B 0.000,C 90.000,E1 70.134} C_DIS
LIN {X -0.068,Y -588.142,Z 1313.181,A 0.000,B 0.000,C 90.000,E1 68.539} C_DIS
LIN {X 0.087,Y -589.239,Z 1313.172,A 0.000,B 0.000,C 90.000,E1 66.922} C_DIS
LIN {X 0.154,Y -590.513,Z 1313.161,A 0.000,B 0.000,C 90.000,E1 65.049} C_DIS
LIN {X 0.127,Y -591.991,Z 1313.150,A 0.000,B 0.000,C 90.000,E1 62.922} C_DIS
LIN {X 0.246,Y -593.600,Z 1313.139,A 0.000,B 0.000,C 90.000,E1 61.051} C_DIS
LIN {X 0.068,Y -595.675,Z 1313.128,A 0.000,B 0.000,C 90.000,E1 58.948} C_DIS
LIN {X 0.053,Y -597.947,Z 1313.116,A 0.000,B 0.000,C 90.000,E1 56.834} C_DIS
LIN {X -0.043,Y -599.631,Z 1313.107,A 0.000,B 0.000,C 90.000,E1 55.261} C_DIS
LIN {X 0.333,Y -600.863,Z 1313.100,A 0.000,B 0.000,C 90.000,E1 53.909} C_DIS
LIN {X -0.108,Y -602.045,Z 1313.092,A 0.000,B 0.000,C 90.000,E1 52.637} C_DIS
LIN {X -0.170,Y -603.103,Z 1313.085,A 0.000,B 0.000,C 90.000,E1 51.331} C_DIS
LIN {X 0.211,Y -604.355,Z 1313.075,A 0.000,B 0.000,C 90.000,E1 49.461} C_DIS
LIN {X 0.059,Y -604.751,Z 1313.071,A 0.000,B 0.000,C 90.000,E1 48.690} C_DIS
LIN {X -0.088,Y -604.983,Z 1313.066,A 0.000,B 0.000,C 90.000,E1 47.919} C_DIS
LIN {X 0.282,Y -605.213,Z 1313.056,A 0.000,B 0.000,C 90.000,E1 46.053} C_DIS
LIN {X -0.066,Y -605.262,Z 1313.050,A 0.000,B 0.000,C 90.000,E1 45.040} C_DIS
LIN {X -0.414,Y -605.127,Z 1313.044,A 0.000,B 0.000,C 90.000,E1 44.028} C_DIS
LIN {X -0.096,Y -604.722,Z 1313.037,A 0.000,B 0.000,C 90.000,E1 42.690} C_DIS
LIN {X -0.192,Y -604.335,Z 1313.030,A 0.000,B 0.000,C 90.000,E1 41.391} C_DIS
LIN {X -0.089,Y -603.873,Z 1313.024,A 0.000,B 0.000,C 90.000,E1 40.334} C_DIS
LIN {X -0.207,Y -603.274,Z 1313.017,A 0.000,B 0.000,C 90.000,E1 39.036} C_DIS
LIN {X -0.034,Y -602.628,Z 1313.011,A 0.000,B 0.000,C 90.000,E1 37.971} C_DIS
LIN {X 0.252,Y -601.926,Z 1313.007,A 0.000,B 0.000,C 90.000,E1 37.156} C_DIS
LIN {X -0.071,Y -600.793,Z 1313.001,A 0.000,B 0.000,C 90.000,E1 36.137} C_DIS
LIN {X -0.036,Y -598.861,Z 1312.993,A 0.000,B 0.000,C 90.000,E1 34.818} C_DIS
LIN {X -0.260,Y -596.964,Z 1312.988,A 0.000,B 0.000,C 90.000,E1 33.785} C_DIS
LIN {X -0.008,Y -594.698,Z 1312.982,A 0.000,B 0.000,C 90.000,E1 32.704} C_DIS
LIN {X -0.184,Y -592.796,Z 1312.977,A 0.000,B 0.000,C 90.000,E1 31.926} C_DIS
LIN {X -0.085,Y -591.300,Z 1312.974,A 0.000,B 0.000,C 90.000,E1 31.386} C_DIS
LIN {X -0.111,Y -588.844,Z 1312.970,A 0.000,B 0.000,C 90.000,E1 30.590} C_DIS
LIN {X -0.159,Y -585.934,Z 1312.965,A 0.000,B 0.000,C 90.000,E1 29.795} C_DIS
LIN {X -0.114,Y -583.811,Z 1312.963,A 0.000,B 0.000,C 90.000,E1 29.255} C_DIS
LIN {X 0.013,Y -580.223,Z 1312.958,A 0.000,B 0.000,C 90.000,E1 28.437} C_DIS
LIN {X 0.015,Y -577.649,Z 1312.955,A 0.000,B 0.000,C 90.000,E1 27.897} C_DIS
LIN {X 0.157,Y -574.101,Z 1312.951,A 0.000,B 0.000,C 90.000,E1 27.206} C_DIS
LIN {X 0.021,Y -570.263,Z 1312.948,A 0.000,B 0.000,C 90.000,E1 26.539} C_DIS
LIN {X 0.102,Y -566.139,Z 1312.944,A 0.000,B 0.000,C 90.000,E1 25.848} C_DIS
LIN {X 0.150,Y -561.590,Z 1312.940,A 0.000,B 0.000,C 90.000,E1 25.155} C_DIS
LIN {X -0.145,Y -558.712,Z 1312.938,A 0.000,B 0.000,C 90.000,E1 24.771} C_DIS
LIN {X -0.270,Y -552.370,Z 1312.933,A 0.000,B 0.000,C 90.000,E1 23.951} C_DIS
LIN {X 0.161,Y -546.802,Z 1312.929,A 0.000,B 0.000,C 90.000,E1 23.206} C_DIS
LIN {X 0.268,Y -538.288,Z 1312.924,A 0.000,B 0.000,C 90.000,E1 22.206} C_DIS
LIN {X -0.092,Y -531.880,Z 1312.920,A 0.000,B 0.000,C 90.000,E1 21.535} C_DIS
LIN {X -0.088,Y -522.787,Z 1312.914,A 0.000,B 0.000,C 90.000,E1 20.556} C_DIS
LIN {X 0.041,Y -512.331,Z 1312.908,A 0.000,B 0.000,C 90.000,E1 19.450} C_DIS
LIN {X -0.022,Y -502.783,Z 1312.903,A 0.000,B 0.000,C 90.000,E1 18.489} C_DIS
LIN {X 0.150,Y -490.499,Z 1312.896,A 0.000,B 0.000,C 90.000,E1 17.275} C_DIS
LIN {X 0.165,Y -484.955,Z 1312.893,A 0.000,B 0.000,C 90.000,E1 16.732} C_DIS
LIN {X -0.080,Y -476.213,Z 1312.889,A 0.000,B 0.000,C 90.000,E1 15.953} C_DIS
LIN {X 0.014,Y -465.946,Z 1312.883,A 0.000,B 0.000,C 90.000,E1 15.009} C_DIS
LIN {X 0.133,Y -444.009,Z 1312.872,A 0.000,B 0.000,C 90.000,E1 12.939} C_DIS
LIN {X 0.065,Y -426.803,Z 1312.862,A 0.000,B 0.000,C 90.000,E1 11.186} C_DIS
LIN {X 0.066,Y -409.668,Z 1312.852,A 0.000,B 0.000,C 90.000,E1 9.321} C_DIS
LIN {X -0.145,Y -400.005,Z 1312.846,A 0.000,B 0.000,C 90.000,E1 8.276} C_DIS
LIN {X -0.110,Y -398.608,Z 1312.845,A 0.000,B 0.000,C 90.000,E1 8.106} C_DIS
LIN {X 0.145,Y -395.447,Z 1312.842,A 0.000,B 0.000,C 90.000,E1 7.587} C_DIS
LIN {X 0.108,Y -395.465,Z 1312.842,A 0.000,B 0.000,C 90.000,E1 7.587} C_DIS
LIN {X 0.171,Y -396.031,Z 1312.842,A 0.000,B 0.000,C 90.000,E1 7.473} C_DIS
LIN {X -0.123,Y -398.952,Z 1312.840,A 0.000,B 0.000,C 90.000,E1 7.239} C_DIS
LIN {X 0.120,Y -404.811,Z 1312.838,A 0.000,B 0.000,C 90.000,E1 6.777} C_DIS
LIN {X -0.155,Y -412.810,Z 1312.835,A 0.000,B 0.000,C 90.000,E1 6.315} C_DIS
LIN {X 0.095,Y -420.839,Z 1312.832,A 0.000,B 0.000,C 90.000,E1 5.739} C_DIS
LIN {X 0.182,Y -426.952,Z 1312.829,A 0.000,B 0.000,C 90.000,E1 5.277} C_DIS
LIN {X 0.014,Y -431.588,Z 1312.828,A 0.000,B 0.000,C 90.000,E1 4.935} C_DIS
LIN {X -0.041,Y -439.129,Z 1312.824,A 0.000,B 0.000,C 90.000,E1 4.302} C_DIS
LIN {X 0.067,Y -443.531,Z 1312.822,A 0.000,B 0.000,C 90.000,E1 3.898} C_DIS
LIN {X 0.018,Y -450.887,Z 1312.818,A 0.000,B 0.000,C 90.000,E1 3.212} C_DIS
LIN {X -0.199,Y -458.077,Z 1312.814,A 0.000,B 0.000,C 90.000,E1 2.522} C_DIS
LIN {X -0.039,Y -462.192,Z 1312.812,A 0.000,B 0.000,C 90.000,E1 2.064} C_DIS
LIN {X -0.018,Y -467.361,Z 1312.808,A 0.000,B 0.000,C 90.000,E1 1.489} C_DIS
LIN {X 0.073,Y -472.447,Z 1312.805,A 0.000,B 0.000,C 90.000,E1 0.859} C_DIS
LIN {X -0.207,Y -478.387,Z 1312.801,A 0.000,B 0.000,C 90.000,E1 0.115} C_DIS
LIN {X 0.134,Y -483.745,Z 1312.796,A 0.000,B 0.000,C 90.000,E1 359.312} C_DIS
LIN {X -0.072,Y -488.668,Z 1312.792,A 0.000,B 0.000,C 90.000,E1 358.568} C_DIS
LIN {X -0.218,Y -493.256,Z 1312.788,A 0.000,B 0.000,C 90.000,E1 357.822} C_DIS
LIN {X 0.154,Y -497.566,Z 1312.784,A 0.000,B 0.000,C 90.000,E1 357.020} C_DIS
LIN {X 0.095,Y -501.527,Z 1312.779,A 0.000,B 0.000,C 90.000,E1 356.274} C_DIS
LIN {X 0.073,Y -505.250,Z 1312.775,A 0.000,B 0.000,C 90.000,E1 355.527} C_DIS
LIN {X -0.112,Y -508.029,Z 1312.772,A 0.000,B 0.000,C 90.000,E1 354.951} C_DIS
LIN {X -0.120,Y -512.619,Z 1312.766,A 0.000,B 0.000,C 90.000,E1 353.913} C_DIS
LIN {X -0.045,Y -515.647,Z 1312.762,A 0.000,B 0.000,C 90.000,E1 353.166} C_DIS
LIN {X -0.181,Y -518.875,Z 1312.757,A 0.000,B 0.000,C 90.000,E1 352.299} C_DIS
LIN {X 0.231,Y -521.830,Z 1312.752,A 0.000,B 0.000,C 90.000,E1 351.376} C_DIS
LIN {X 0.235,Y -523.631,Z 1312.749,A 0.000,B 0.000,C 90.000,E1 350.792} C_DIS
LIN {X 0.197,Y -526.972,Z 1312.743,A 0.000,B 0.000,C 90.000,E1 349.634} C_DIS
LIN {X -0.249,Y -529.202,Z 1312.738,A 0.000,B 0.000,C 90.000,E1 348.814} C_DIS
LIN {X -0.114,Y -531.812,Z 1312.731,A 0.000,B 0.000,C 90.000,E1 347.645} C_DIS
LIN {X 0.129,Y -533.488,Z 1312.727,A 0.000,B 0.000,C 90.000,E1 346.756} C_DIS
LIN {X -0.249,Y -534.901,Z 1312.722,A 0.000,B 0.000,C 90.000,E1 345.936} C_DIS
LIN {X 0.034,Y -536.158,Z 1312.717,A 0.000,B 0.000,C 90.000,E1 345.046} C_DIS
LIN {X 0.137,Y -536.861,Z 1312.714,A 0.000,B 0.000,C 90.000,E1 344.464} C_DIS
LIN {X 0.124,Y -537.827,Z 1312.708,A 0.000,B 0.000,C 90.000,E1 343.323} C_DIS
LIN {X -0.082,Y -538.370,Z 1312.703,A 0.000,B 0.000,C 90.000,E1 342.489} C_DIS
LIN {X -0.117,Y -538.542,Z 1312.698,A 0.000,B 0.000,C 90.000,E1 341.638} C_DIS
LIN {X -0.106,Y -538.301,Z 1312.692,A 0.000,B 0.000,C 90.000,E1 340.496} C_DIS
LIN {X 0.045,Y -537.754,Z 1312.687,A 0.000,B 0.000,C 90.000,E1 339.625} C_DIS
LIN {X 0.008,Y -536.967,Z 1312.682,A 0.000,B 0.000,C 90.000,E1 338.773} C_DIS
LIN {X -0.045,Y -535.974,Z 1312.677,A 0.000,B 0.000,C 90.000,E1 337.922} C_DIS
LIN {X -0.117,Y -535.054,Z 1312.674,A 0.000,B 0.000,C 90.000,E1 337.358} C_DIS
LIN {X -0.194,Y -533.808,Z 1312.671,A 0.000,B 0.000,C 90.000,E1 336.794} C_DIS
LIN {X 0.010,Y -533.372,Z 1312.669,A 0.000,B 0.000,C 90.000,E1 336.485} C_DIS
LIN {X 0.116,Y -531.229,Z 1312.665,A 0.000,B 0.000,C 90.000,E1 335.613} C_DIS
LIN {X -0.283,Y -528.784,Z 1312.660,A 0.000,B 0.000,C 90.000,E1 334.793} C_DIS
LIN {X 0.244,Y -523.236,Z 1312.650,A 0.000,B 0.000,C 90.000,E1 332.999} C_DIS
LIN {X 0.053,Y -518.471,Z 1312.642,A 0.000,B 0.000,C 90.000,E1 331.563} C_DIS
LIN {X 0.124,Y -514.350,Z 1312.636,A 0.000,B 0.000,C 90.000,E1 330.383} C_DIS
LIN {X 0.306,Y -510.435,Z 1312.630,A 0.000,B 0.000,C 90.000,E1 329.331} C_DIS
LIN {X 0.123,Y -504.223,Z 1312.622,A 0.000,B 0.000,C 90.000,E1 327.867} C_DIS
LIN {X 0.044,Y -499.905,Z 1312.616,A 0.000,B 0.000,C 90.000,E1 326.834} C_DIS
LIN {X 0.080,Y -496.646,Z 1312.611,A 0.000,B 0.000,C 90.000,E1 325.928} C_DIS
LIN {X 0.221,Y -494.953,Z 1312.607,A 0.000,B 0.000,C 90.000,E1 325.308} C_DIS
LIN {X 0.034,Y -493.286,Z 1312.603,A 0.000,B 0.000,C 90.000,E1 324.436} C_DIS
LIN {X -0.173,Y -491.102,Z 1312.592,A 0.000,B 0.000,C 90.000,E1 322.637} C_DIS
LIN {X 0.207,Y -490.266,Z 1312.589,A 0.000,B 0.000,C 90.000,E1 321.984} C_DIS
LIN {X -0.107,Y -489.246,Z 1312.586,A 0.000,B 0.000,C 90.000,E1 321.412} C_DIS
LIN {X 0.039,Y -488.621,Z 1312.584,A 0.000,B 0.000,C 90.000,E1 321.090} C_DIS
LIN {X -0.123,Y -487.864,Z 1312.582,A 0.000,B 0.000,C 90.000,E1 320.803} C_DIS
LIN {X 0.023,Y -486.887,Z 1312.581,A 0.000,B 0.000,C 90.000,E1 320.481} C_DIS
LIN {X -0.215,Y -486.239,Z 1312.580,A 0.000,B 0.000,C 90.000,E1 320.356} C_DIS
LIN {X -0.143,Y -485.363,Z 1312.579,A 0.000,B 0.000,C 90.000,E1 320.194} C_DIS
LIN {X 0.054,Y -482.399,Z 1312.577,A 0.000,B 0.000,C 90.000,E1 319.865} C_DIS
LIN {X 0.116,Y -460.434,Z 1312.564,A 0.000,B 0.000,C 90.000,E1 317.553} C_DIS
LIN {X 0.036,Y -440.603,Z 1312.551,A 0.000,B 0.000,C 90.000,E1 315.202} C_DIS
LIN {X 0.207,Y -422.189,Z 1312.537,A 0.000,B 0.000,C 90.000,E1 312.690} C_DIS
LIN {X -0.107,Y -405.544,Z 1312.523,A 0.000,B 0.000,C 90.000,E1 310.172} C_DIS
LIN {X 0.039,Y -390.547,Z 1312.509,A 0.000,B 0.000,C 90.000,E1 307.523} C_DIS
LIN {X -0.020,Y -388.140,Z 1312.506,A 0.000,B 0.000,C 90.000,E1 307.076} C_DIS
LIN {X -0.058,Y -388.139,Z 1312.506,A 0.000,B 0.000,C 90.000,E1 307.076} C_DIS
LIN {X -0.109,Y -391.148,Z 1312.493,A 0.000,B 0.000,C 90.000,E1 304.692} C_DIS
LIN {X 0.057,Y -392.156,Z 1312.485,A 0.000,B 0.000,C 90.000,E1 303.245} C_DIS
LIN {X 0.244,Y -396.866,Z 1312.459,A 0.000,B 0.000,C 90.000,E1 298.615} C_DIS
LIN {X -0.202,Y -397.299,Z 1312.455,A 0.000,B 0.000,C 90.000,E1 297.975} C_DIS
LIN {X -0.115,Y -401.619,Z 1312.426,A 0.000,B 0.000,C 90.000,E1 292.695} C_DIS
LIN {X 0.005,Y -404.687,Z 1312.395,A 0.000,B 0.000,C 90.000,E1 287.094} C_DIS
LIN {X -0.193,Y -404.734,Z 1312.389,A 0.000,B 0.000,C 90.000,E1 286.079} C_DIS
LIN {X -0.002,Y -406.117,Z 1312.364,A 0.000,B 0.000,C 90.000,E1 281.535} C_DIS
LIN {X 0.018,Y -405.949,Z 1312.360,A 0.000,B 0.000,C 90.000,E1 280.838} C_DIS
LIN {X 0.091,Y -405.687,Z 1312.333,A 0.000,B 0.000,C 90.000,E1 275.967} C_DIS
LIN {X 0.128,Y -403.478,Z 1312.304,A 0.000,B 0.000,C 90.000,E1 270.745} C_DIS
LIN {X 0.095,Y -403.268,Z 1312.302,A 0.000,B 0.000,C 90.000,E1 270.401} C_DIS
LIN {X -0.123,Y -398.897,Z 1312.271,A 0.000,B 0.000,C 90.000,E1 264.837} C_DIS
LIN {X 0.171,Y -393.363,Z 1312.244,A 0.000,B 0.000,C 90.000,E1 259.859} C_DIS
LIN {X 0.093,Y -392.800,Z 1312.240,A 0.000,B 0.000,C 90.000,E1 259.162} C_DIS
LIN {X -0.202,Y -386.345,Z 1312.214,A 0.000,B 0.000,C 90.000,E1 254.574} C_DIS
LIN {X 0.132,Y -385.237,Z 1312.208,A 0.000,B 0.000,C 90.000,E1 253.449} C_DIS
LIN {X 0.152,Y -384.709,Z 1312.206,A 0.000,B 0.000,C 90.000,E1 253.087} C_DIS
LIN {X 0.010,Y -377.931,Z 1312.182,A 0.000,B 0.000,C 90.000,E1 248.773} C_DIS
LIN {X 0.092,Y -376.198,Z 1312.174,A 0.000,B 0.000,C 90.000,E1 247.305} C_DIS
LIN {X -0.063,Y -373.548,Z 1312.166,A 0.000,B 0.000,C 90.000,E1 245.869} C_DIS
LIN {X 0.036,Y -366.949,Z 1312.141,A 0.000,B 0.000,C 90.000,E1 241.435} C_DIS
LIN {X -0.112,Y -365.984,Z 1312.137,A 0.000,B 0.000,C 90.000,E1 240.717} C_DIS
